# B&R Automation Studio project vibratorControlWithCurrentController (part 12)

#### producing.st
```iecst
ACTION producing:

	CASE em.state OF

		STATE_STOPPED:

			interface.status.ready 	:= FALSE;
			interface.status.active := TRUE; // need to tell wing when we are active. (otherwise wing start too fast and this task is stuck in STATE_ACTIVATING doing boot)

			em.cmd.sc 				:= TRUE;

		STATE_RESETTING:

			em.cmd.sc := TRUE;

		STATE_IDLE:
			interface.status.ready := TRUE;
			em.cmd.sc := TRUE;

		STATE_STARTING:

			interface.status.ready 									:= TRUE;
			interface.cmd.start										:= FALSE;
			interface.status.readyForStatusChange 					:= TRUE;
			this.cycleTime 											:= 0;
			em.cmd.sc 												:= TRUE;

		STATE_EXECUTE:

			CASE em.substate OF
				0: // H010 (Initialisation) + H020 (FM Start)
					em.cmd.sc := TRUE;
					interface.status.ready	:= TRUE;

					em.description := 'waiting for start command';
					IF interface.cmd.start THEN
						this.calculateCycletime := TRUE;
						IF interface.parameter.brickStatus = BRICK_STATUS_OK THEN
							this.MTDataStatistics_Real.Enable				:= TRUE;
							this.MTDataStatistics_Real.MovingWindowLength 	:= 10;
							this.MTDataStatistics_Real.In 					:= this.cycleTimeReal / 1000;
							this.MTDataStatistics_Real();
							this.cycleTimeReal := 0;
							IF this.MTDataStatistics_Real.Mean <> 0 THEN
								this.hmi.realMeanOutput := 60000 / this.MTDataStatistics_Real.Mean;
							END_IF
						END_IF

						// calculate cycletime here
						interface.cmd.start 						:= FALSE;
						interface.status.ready 						:= FALSE;
						this.time.elapsed							:= 0;
						this.time.maximum							:= interface.parameter.fallTime;
						gBottomFlapInterface.parameter.brickStatus 	:= interface.parameter.brickStatus;
						gBottomFlapInterface.cmd.brickStatusReady	:= TRUE;
						this.middleFlapTime 						:= 0;
						em.substate 								:= 40;
					ELSIF interface.cmd.manuelMode THEN
						em.substate := 1000;
					END_IF

				40: // H040 (FB Ready)
					em.description := 'waiting for bottom flap ready1 or ready2';

					this.time.elapsed := this.time.elapsed + em.status.cycleTime;

					IF gBottomFlapInterface.status.ready1 THEN
						interface.status.readyForStatusChange 		:= FALSE;
						gBottomFlapInterface.cmd.brickStatusReady	:= FALSE;
						gBottomFlapInterface.cmd.start1	:= TRUE;
						//em.cmd.sc := FALSE;
					END_IF

					// Wait FallTime before giving start2 (ok to give start1 before)
					IF gBottomFlapInterface.status.ready2 THEN
						em.cmd.sc := FALSE;
						this.flap.open := TRUE;
						this.cycleTimeTheoretical := 0;
						this.middleFlapTime := this.middleFlapTime + em.status.cycleTime;
						em.substate 			:= 70;
					END_IF

				70: // H070 (Open FM)
					em.description 				:= 'waiting for flap to be open';

					this.middleFlapTime := this.middleFlapTime + em.status.cycleTime;

					IF this.flap.error THEN
						this.alarm.openTooLong.active := TRUE;
						this.previousState := em.substate;
						em.substate := 700; // Error state in execute
					ELSIF this.flap.position = FLAP_OPEN THEN
						this.time.elapsed				:= 0;
						this.time.maximum				:= interface.parameter.openTime;
						gBottomFlapInterface.cmd.start2 := TRUE;
						interface.status.lastCycleTime 	:= UDINT_TO_REAL(this.middleFlapTime);
						interface.status.openCloseTime := this.cycleTimeTheoretical;
						em.substate 					:= 75;
					END_IF

				75: // H075
					em.description := 'waiting for opening time';

					this.middleFlapTime := this.middleFlapTime + em.status.cycleTime;
					this.time.elapsed	:= this.time.elapsed + em.status.cycleTime;

					IF this.time.elapsed >= this.time.maximum THEN
						this.flap.close := TRUE;
						em.substate := 80;
					END_IF

				80: // H080 (Close FM)
					em.description 				:= 'waiting for flap to be closed';

					this.middleFlapTime := this.middleFlapTime + em.status.cycleTime;

					IF this.flap.error THEN
						this.alarm.closeTooLong.active := TRUE;
						this.previousState := em.substate;
						em.substate := 700; // Error state in execute
					ELSIF this.flap.position = FLAP_CLOSED THEN
						interface.status.ready	:= TRUE;
						// Save open/close time in service menu (better than writing it cyclically).
						this.flapTest.openTime := this.flap.openTimeAfterChangeover;
						this.flapTest.closingTime := this.flap.closingTimeAfterChangeover;
						this.flapTest.openTimeOK := this.flapTest.openTime >= 210 AND this.flapTest.openTime <= 230;
						this.flapTest.closingTimeOK := this.flapTest.closingTime >= 210 AND this.flapTest.closingTime <= 230;
						this.cycleTime 			:= 0;
						this.hmi.portionCycleTime := UDINT_TO_REAL(this.middleFlapTime+gUpperFlapInterface.status.lastCycleTime)/1000;
						em.substate 			:= 0;
					END_IF

					(**** ERROR handling in EXECUTE ****)

				700:
					interface.cmd.runFlapContinuously	:= FALSE;
					interface.cmd.open					:= FALSE;
					interface.cmd.manuelMode			:= FALSE;

					IF NOT this.flap.error THEN
						this.flap.close := TRUE;
						em.substate := 710;
					ELSE
						this.flap.resetError := TRUE;
					END_IF

				710:
					em.description := 'Wait for flap to close - if not still continue. We cant be stuck in "SUSPENDING"';

					IF this.flap.error THEN
						this.time.elapsed := 0;
						em.substate := 720;
					ELSIF this.flap.position = FLAP_CLOSED THEN
						this.time.elapsed := 0;
						em.substate := 720;
					END_IF

				720:
					em.description := 'Wait for alarm acknowledge';

					this.time.elapsed := this.time.elapsed + em.status.cycleTime;

					IF this.time.elapsed >= 500000 THEN //500ms
						this.time.elapsed := 0;
						IF NOT MpAlarmXCheckReaction(mpAlarmXCore,'abortMain') THEN
							em.substate := 730; // "UNSUSPENDING"
						END_IF
					END_IF

				730:
					IF NOT this.flap.error THEN
						brsmemset(ADR(this.alarm), 0, SIZEOF(this.alarm));
						this.alarm.closeTooLong.name := 'middleFlapCloseTooLong';
						this.alarm.openTooLong.name := 'middleFlapOpenTooLong';
						this.flap.close := TRUE;
						em.substate := 740;
					ELSE
						this.flap.resetError := TRUE;
					END_IF

				740:
					em.description := 'Wait for flap to close -> if not go back and try again ';

					IF this.flap.error THEN
						em.substate := 730; // Try again (we MUST close flap before we return)
					ELSIF this.flap.position = FLAP_CLOSED THEN
						em.substate := 750;
					END_IF

				750:
					em.description := 'Recover to "previousState"';

					CASE this.previousState OF

						70: // Error opening
							em.cmd.sc := FALSE;
							this.flap.open := TRUE;
							this.cycleTimeTheoretical := 0;
							em.substate 			:= 70;

						80: // Error closing
							this.flap.close := TRUE;
							em.substate := 80;

						1000:
							em.substate := 0;

					END_CASE

					(**** Manuel mode ****)

				1000:
					testing;
					IF this.flap.error THEN
						// Stop testing and go in execute error state.
						this.previousState := em.substate;
						this.test.state := 0;

						em.substate := 700;
					END_IF

			END_CASE

			IF gMainInterface.status.state = STATE_EXECUTE THEN
				// calculate throughput cycletime
				this.cycleTime := this.cycleTime + UDINT_TO_REAL(em.status.cycleTime);
				this.cycleTimeReal := this.cycleTimeReal + UDINT_TO_REAL(em.status.cycleTime);
			ELSE
				this.MTDataStatistics_Real.Enable := FALSE;
				this.MTDataStatistics_Real();
				this.calculateCycletime := FALSE;
				this.cycleTime := 0;
				this.cycleTimeReal := 0;
				this.hmi.realMeanOutput := 0;
			END_IF

			this.cycleTimeTheoretical := this.cycleTimeTheoretical + em.status.cycleTime;

		STATE_COMPLETING:

			em.description := 'waiting for bottom flap ready2 to be ready';

			CASE em.substate OF

				0:
					// Determine if big or small brick from capcon teach integral
					IF gCapconInterface.status.teachIntegral > ELEMENT_SIZE_LIMIT AND gCapconInterface.status.teachingDone THEN
						this.ItemSize := Large;
					ELSE
						this.ItemSize := Small;
					END_IF

					em.substate := 10;

				10:
					IF gBottomFlapInterface.status.ready2 THEN
						gBeltInterface.cmd.stopDoingEmpty := FALSE;
						em.cmd.sc := TRUE;
					END_IF

			END_CASE

			em.setup.reactTo := BRDK_EM_REACT_TO_ALL;

		STATE_COMPLETE:

			CASE em.substate OF

				0:
					em.description 		:= 'empty or small items empty';

					IF this.ItemSize=Small THEN
						this.time.maximum := TIME_EMPTY_SMALL_ITEM;
						em.cmd.sc := FALSE;
						em.substate := 5;
					ELSE
						this.flap.open := TRUE;
						em.substate := 10;
						em.cmd.sc := TRUE;
					END_IF

				5:
					interface.status.ready := TRUE;
					em.description 		:= 'waiting for empty small items time or empty finished';
					this.time.elapsed	:= this.time.elapsed + em.status.cycleTime;

					IF this.time.elapsed >= this.time.maximum OR gMainInterface.status.state <> STATE_COMPLETING THEN
						interface.status.busy 	:= TRUE;
						this.time.elapsed 	:= 0;
						this.flap.open := TRUE;
						em.cmd.sc := FALSE;
						gBeltInterface.cmd.stopDoingEmpty := TRUE;
						em.substate 			:= 10;
					END_IF

					IF this.time.elapsed >= (this.time.maximum-400000) THEN
						// Signal belt and vibrator to stop 0.4s before opening flap.
						gBeltInterface.cmd.stopDoingEmpty := TRUE;
					END_IF

				10: // H820 (FM open)
					em.description 			:= 'waiting for flap to be open';

					IF this.flap.error THEN
						this.alarm.openTooLong.active := TRUE;
						this.previousState := em.substate;
						em.substate := 700; // Error state in execute
					ELSIF this.flap.position = FLAP_OPEN THEN
						this.time.elapsed				:= 0;
						this.time.maximum				:= 1000000; // 1s. be open for a longer time because a lot of bricks is falling and we dont want to pierce them.
						em.cmd.sc := TRUE;

						IF this.ItemSize=Small THEN
							em.substate 					:= 20;
						ELSE
							em.substate 					:= 40;
						END_IF

					END_IF

				20: //
					em.description 		:= 'waiting for opening time';
					this.time.elapsed	:= this.time.elapsed + em.status.cycleTime;

					IF this.time.elapsed >= this.time.maximum THEN
						this.flap.close := TRUE;
						em.cmd.sc := FALSE;
						interface.status.busy 			:= FALSE;
						em.substate 					:= 30;
					END_IF

				30: // H830 (FM close)
					em.description 		:= 'waiting for flap to be closed';

					IF this.flap.error THEN
						this.alarm.closeTooLong.active := TRUE;
						this.previousState := em.substate;
						em.substate := 700; // Error state in execute
					ELSIF this.flap.position = FLAP_CLOSED THEN
						interface.status.ready	:= TRUE;
						gBeltInterface.cmd.stopDoingEmpty := FALSE;
						this.flapTest.openTime := this.flap.openTimeAfterChangeover;
						this.flapTest.closingTime := this.flap.closingTimeAfterChangeover;
						this.flapTest.openTimeOK := this.flapTest.openTime >= 210 AND this.flapTest.openTime <= 230;
						this.flapTest.closingTimeOK := this.flapTest.closingTime >= 210 AND this.flapTest.closingTime <= 230;
						em.substate 			:= 0;
					END_IF

				40:
					em.description 		:= 'Emptying machine';
					interface.status.ready := TRUE;

						(**** ERROR handling in COMPLETE ****)

				700:
					interface.cmd.runFlapContinuously	:= FALSE;
					interface.cmd.open					:= FALSE;
					interface.cmd.manuelMode			:= FALSE;

					IF NOT this.flap.error THEN
						this.flap.close := TRUE;
						em.substate := 710;
					ELSE
						this.flap.resetError := TRUE;
					END_IF

				710:
					em.description := 'Wait for flap to close - if not still continue. We cant be stuck in "SUSPENDING"';

					IF this.flap.error THEN
						this.time.elapsed := 0;
						em.substate := 720;
					ELSIF this.flap.position = FLAP_CLOSED THEN
						this.time.elapsed := 0;
						em.substate := 720;
					END_IF

				720:
					em.description := 'Wait for alarm acknowledge';

					this.time.elapsed := this.time.elapsed + em.status.cycleTime;

					IF this.time.elapsed >= 500000 THEN //500ms
						this.time.elapsed := 0;
						IF NOT MpAlarmXCheckReaction(mpAlarmXCore,'abortMain') THEN
							em.substate := 730; // "UNSUSPENDING"
						END_IF
					END_IF

				730:
					IF NOT this.flap.error THEN
						brsmemset(ADR(this.alarm), 0, SIZEOF(this.alarm));
						this.alarm.closeTooLong.name := 'middleFlapCloseTooLong';
						this.alarm.openTooLong.name := 'middleFlapOpenTooLong';
						this.flap.close := TRUE;
						em.substate := 740;
					ELSE
						this.flap.resetError := TRUE;
					END_IF

				740:
					em.description := 'Wait for flap to close -> if not go back and try again ';

					IF this.flap.error THEN
						em.substate := 730; // Try again (we MUST close flap before we return)
					ELSIF this.flap.position = FLAP_CLOSED THEN
						em.substate := 750;
					END_IF

				750:
					em.description := 'Recover to "previousState"';

					CASE this.previousState OF

						10: // Error opening
							em.substate 			:= 0;

						30: // Error closing
							this.time.elapsed := 0;
							this.time.maximum := interface.parameter.openTime;
							em.substate := 20;

					END_CASE

		END_CASE

			gBottomFlapInterface.cmd.start1 := em.cmd.sc;

	STATE_ABORTED, STATE_SUSPENDED:
			em.description := 'waiting for wing to start';
			em.cmd.sc := TRUE;

	STATE_STOPPING, STATE_ABORTING, STATE_SUSPENDING:

			CASE em.substate OF

				0:
					em.description 				:= 'Clear status and close flap';
					interface.status.ready 					:= FALSE;
					interface.status.readyForStatusChange 	:= FALSE;
					interface.cmd.start 					:= FALSE;
					this.hw.do_open 		:= FALSE;
					interface.cmd.runFlapContinuously	:= FALSE;
					interface.cmd.open					:= FALSE;
					interface.cmd.manuelMode			:= FALSE;
					gBeltInterface.cmd.stopDoingEmpty := FALSE;

					IF NOT this.flap.error THEN
						this.flap.close := TRUE;
						em.substate := 10;
					ELSE
						this.flap.resetError := TRUE;
					END_IF

				10:
					em.description := 'Wait for flap to close';

					IF this.flap.error THEN
						em.substate := 20;
					ELSIF this.flap.position = FLAP_CLOSED THEN
						em.substate := 20;
					END_IF

				20:
					em.cmd.sc := TRUE;

			END_CASE

	STATE_CLEARING, STATE_UNSUSPENDING:
		em.description := 'waiting for flap error reset';

			CASE em.substate OF

				0:
					IF NOT this.flap.error THEN
						brsmemset(ADR(this.alarm), 0, SIZEOF(this.alarm));
						this.alarm.closeTooLong.name := 'middleFlapCloseTooLong';
						this.alarm.openTooLong.name := 'middleFlapOpenTooLong';
						this.flap.close := TRUE;
						em.substate := 10;
					ELSE
						this.flap.resetError := TRUE;
					END_IF

				10:
					em.description := 'Wait for flap to close';

					IF this.flap.error THEN
						em.substate := 0;
					ELSIF this.flap.position = FLAP_CLOSED THEN
						em.substate := 20;
					END_IF

				20:
					em.description 				:= 'Wait for close of own and neigbourflap';
					em.cmd.sc := TRUE;

			END_CASE

	ELSE
	em.cmd.sc := TRUE;

	END_CASE

END_ACTION
```

#### alarm.st
```iecst
ACTION alarm:

	// Open Time Too Long

	IF this.alarm.openTooLong.active AND NOT this.alarm.openTooLong.oldActive THEN
		this.alarm.openTooLong.instanceID := MpAlarmXSet(mpAlarmXCore, this.alarm.openTooLong.name);
	END_IF
	this.alarm.openTooLong.oldActive := this.alarm.openTooLong.active;

	// Close Time Too Long

	IF this.alarm.closeTooLong.active AND NOT this.alarm.closeTooLong.oldActive THEN
		this.alarm.closeTooLong.instanceID := MpAlarmXSet(mpAlarmXCore, this.alarm.closeTooLong.name);
	END_IF
	this.alarm.closeTooLong.oldActive := this.alarm.closeTooLong.active;

END_ACTION
```

#### middleFlap.st - Init, cyclic, exit code
```iecst
PROGRAM _INIT

	em.setup.name 			:= 'middleFlap';
	em.setup.parent.name 	:= 'wing';
	em.setup.reactTo 		:= BRDK_EM_REACT_TO_ALL;

	setupPointers;

	this.alarm.closeTooLong.name := 'middleFlapCloseTooLong';
	this.alarm.openTooLong.name := 'middleFlapOpenTooLong';

END_PROGRAM

PROGRAM _CYCLIC

	setupPointers;
	ioMappingInput;

	// setup flap function block
	this.flap.enable				:= TRUE;
	this.flap.cycleTime				:= em.status.cycleTime;
	this.flap.flapTime				:= interface.parameter.flapTime;
	this.flap.di_changeover 		:= this.hw.di_changeover;
	this.flap.simulation := gWingInterface.parameter.simulation;

	CASE em.mode OF
		MODE_PRODUCING,MODE_EMPTY: producing;
		MODE_MANUAL: testing;	// mode for testing flaps manually.
		ELSE em.cmd.sc := TRUE;
	END_CASE

	this.hw.do_open := this.flap.do_open;

	alarm;

	em();
	this.flap();

	// FAT test
	CASE testStateFAT OF

		0:
			IF interface.cmd.wingTestManual THEN
				// Only execute if flap is closed
				IF this.hw.do_open=FALSE THEN
					interface.status.testResultFAT := FALSE; // reset result
					testStateFAT := 10;
				END_IF

			END_IF

		10:
			//wait 1s so flaps are closed before we start test.
			this.TON_test.IN := TRUE;
			this.TON_test.PT := T#500ms;
			this.TON_test();

			IF this.TON_test.Q THEN
				this.TON_test.IN := FALSE;
				this.TON_test();

				// Open flap
				this.flap.open := TRUE;
				testStateFAT := 20;
			END_IF

		20:
			IF this.flap.error THEN
				// Test fail
				testStateFAT := 60;
			ELSIF this.flap.position = FLAP_OPEN THEN
				testStateFAT 			:= 30;
			END_IF

		30:
			//wait 1s before closing
			this.TON_test.IN := TRUE;
			this.TON_test.PT := T#500ms;
			this.TON_test();

			IF this.TON_test.Q THEN
				this.TON_test.IN := FALSE;
				this.TON_test();

				// Close flap
				this.flap.close := TRUE;
				testStateFAT := 40;
			END_IF

		40:
			IF this.flap.error THEN
				// Test fail
				testStateFAT := 60;
			ELSIF this.flap.position = FLAP_CLOSED THEN
				testStateFAT 			:= 50;
			END_IF

		50:
			//wait 1s before closing
			this.TON_test.IN := TRUE;
			this.TON_test.PT := T#500ms;
			this.TON_test();

			IF this.TON_test.Q THEN
				this.TON_test.IN := FALSE;
				this.TON_test();

				interface.status.testResultFAT := TRUE; // Good result
				testStateFAT := 60;
			END_IF

		60:
			// Reset error (if any) before finishing test
			this.flap.resetError := this.flap.error;

			IF NOT this.flap.error THEN
				interface.cmd.wingTestManual := FALSE; // signal test done

				// Start next test (we are done here)
				gBottomFlapInterface.cmd.wingTestManual := TRUE;
				testStateFAT := 0;
			END_IF

	END_CASE

END_PROGRAM

PROGRAM _EXIT

END_PROGRAM
```

#### ioMappingInput.st
```iecst
ACTION ioMappingInput:

	IF this.hwWu[0].di_wingUnitActive THEN
		this.flap.WUstepperConnected 	:= TRUE;
		this.flap.positionFromWUstepper	:= this.hwWu[0].flapPosition;
	ELSIF this.hwWu[1].di_wingUnitActive THEN
		this.flap.WUstepperConnected 	:= TRUE;
		this.flap.positionFromWUstepper	:= this.hwWu[1].flapPosition;
	ELSE
		this.flap.WUstepperConnected := FALSE;
	END_IF

END_ACTION
```

#### testing.st
```iecst
ACTION testing:

	this.flapTest.openTime := this.flap.openTimeAfterChangeover;
	this.flapTest.closingTime := this.flap.closingTimeAfterChangeover;
	this.flapTest.openTimeOK := this.flapTest.openTime >= 210 AND this.flapTest.openTime <= 230;
	this.flapTest.closingTimeOK := this.flapTest.closingTime >= 210 AND this.flapTest.closingTime <= 230;

	CASE this.test.state OF

		0:
			IF NOT interface.cmd.manuelMode THEN
				interface.cmd.runFlapContinuously := FALSE;
				em.substate := 0; // go back to 0 (no more manuel mode)
			ELSIF gWingInterface.status.startTestSequence THEN
				interface.cmd.runFlapContinuously := FALSE; // can't run while doing test sequence.
				this.test.state := 10;
			ELSIF interface.cmd.runFlapContinuously THEN
				this.test.state := 60;
			END_IF

			(**** Run sequence ****)

		10:
			IF NOT gWingInterface.status.startTestSequence THEN
				this.test.state := 0;
			ELSIF interface.cmd.open THEN
				this.flap.open := TRUE;
				this.test.state := 20;
			END_IF

		20:

			IF this.flap.error THEN
				this.alarm.openTooLong.active := TRUE;
			ELSIF this.flap.position = FLAP_OPEN THEN
				this.time.elapsed := 0;
				this.test.state := 30;
			END_IF

		30:
			this.time.elapsed := this.time.elapsed + em.status.cycleTime;
			IF this.time.elapsed >= this.flapTest.waitTime THEN
				this.flap.close := TRUE;		// close cmd
				this.test.state := 40;
			END_IF

		40:
			IF this.flap.error THEN
				this.alarm.closeTooLong.active := TRUE;
			ELSIF this.flap.position = FLAP_CLOSED THEN
				this.time.elapsed := 0;
				this.test.state := 50;
			END_IF

		50:
			em.description := 'Wait delay before opening next flap';

			this.time.elapsed := this.time.elapsed + em.status.cycleTime;
			IF this.time.elapsed >= this.flapTest.waitTime THEN
				interface.cmd.open := FALSE;	// Will signal to wing that flap is done with open/close.
				this.test.state := 10;
			END_IF

			(**** Run continously ****)

		60:
			IF NOT interface.cmd.runFlapContinuously THEN
				this.test.state := 0;
			ELSE
				this.flap.open := TRUE;
				this.test.state := 70;
			END_IF

		70:
			IF this.flap.error THEN
				this.alarm.openTooLong.active := TRUE;
			ELSIF this.flap.position = FLAP_OPEN THEN
				this.time.elapsed := 0;
				this.test.state := 80;
			END_IF

		80:
			this.time.elapsed := this.time.elapsed + em.status.cycleTime;
			IF this.time.elapsed >= this.flapTest.waitTime THEN
				this.flap.close := TRUE;		// close cmd
				this.test.state := 90;
			END_IF

		90:
			IF this.flap.error THEN
				this.alarm.closeTooLong.active := TRUE;
			ELSIF this.flap.position = FLAP_CLOSED THEN
				this.time.elapsed := 0;
				this.test.state := 100;
			END_IF

		100:
			this.time.elapsed := this.time.elapsed + em.status.cycleTime;
			IF this.time.elapsed >= this.flapTest.waitTime THEN
				this.test.state := 60;
			END_IF

	END_CASE

END_ACTION
```

#### setupPointers.st
```iecst
ACTION setupPointers:
	interface ACCESS ADR(gMiddleFlapInterface);
END_ACTION
```

#### local.typ - Local data types
```iecst
TYPE
	local_typ : 	STRUCT
		hw : local_hw_typ;
		hwAir : local_hw_typ;
		hwWu : ARRAY[0..1]OF wu20_typ; (*Communication with wing unit*)
		alarm : local_alarm_typ;
		time : local_time_typ;
		flap : legoCM20Flap;
		flapTest : flapTest_typ;
		MTDataStatistics_Real : MTDataStatistics;
		cycleTime : REAL;
		calculateCycletime : BOOL;
		hmi : local_hmi_typ;
		cycleTimeReal : REAL;
		cycleTimeTheoretical : UDINT;
		test : local_test_typ;
		previousState : UINT;
		middleFlapTime : UDINT;
		ItemSize : ITEM_SIZE_enum;
		TON_test : TON;
	END_STRUCT;
	ITEM_SIZE_enum :
		( (*Default large*)
		Large := 0,
		Small := 1
		);
	wu20_typ : 	STRUCT
		flapPosition : DINT; (*4 = open, 8 = closed*)
		di_wingUnitActive : BOOL;
	END_STRUCT;
	local_hmi_typ : 	STRUCT
		realMeanOutput : REAL;
		cycleTimeRaw : REAL;
		portionCycleTime : REAL;
	END_STRUCT;
	local_hw_typ : 	STRUCT
		di_changeover : BOOL;
		do_open : BOOL;
	END_STRUCT;
	local_alarm_typ : 	STRUCT
		openTooLong : gAlarm_struct_typ;
		closeTooLong : gAlarm_struct_typ;
	END_STRUCT;
	flapTest_typ : 	STRUCT
		flapSequenceTest : BOOL; (*Flaps will run in a sequence (usually over night)*)
		openTime : UDINT;
		closingTime : UDINT;
		waitTime : UDINT := 200000;
		alarmOpenTooLong : BOOL;
		alarmCloseTooLong : BOOL;
		openTimeOK : BOOL;
		closingTimeOK : BOOL;
	END_STRUCT;
	local_test_typ : 	STRUCT
		state : USINT;
	END_STRUCT;
END_TYPE
```

#### local.var - Local variables
```iecst
VAR CONSTANT
	ELEMENT_SIZE_LIMIT : REAL := 250000;
	TIME_EMPTY_SMALL_ITEM : UDINT := 20000000; (*20s*)
END_VAR
VAR
	interface : REFERENCE TO gMiddleFlapInterface_typ;
	this : {REDUND_UNREPLICABLE} local_typ;
	em : {REDUND_UNREPLICABLE} brdkEM;
	testStateFAT : USINT;
END_VAR
```

### middleFlapGlobal.var
```iecst
VAR
	gMiddleFlapInterface : gMiddleFlapInterface_typ;
END_VAR
```

### middleFlapGlobal.typ
```iecst
TYPE
	gMiddleFlapInterface_status_typ : 	STRUCT
		ready : BOOL;
		readyForStatusChange : BOOL;
		busy : BOOL;
		waitingForBottomOrCassette : BOOL;
		openCloseTime : UDINT;
		active : BOOL;
		lastCycleTime : REAL;
		testResultFAT : BOOL; (*TRUE=good, FALSE=bad*)
	END_STRUCT;
	gMiddleFlapInterface_para_typ : 	STRUCT
		brickStatus : gFlap_brick_status_typ;
		openTime : UDINT; (*Time the flap stays open*)
		flapTime : UDINT; (*Time that the flap is to open or close*)
		fallTime : UDINT; (*Time that a brick is to fall and be steady*)
		emptySmallItemsTime : UDINT; (*Time for flipping the flap when emptying small items*)
	END_STRUCT;
	gMiddleFlapInterface_cmd_typ : 	STRUCT
		start : BOOL;
		smallBrick : BOOL;
		updateStatistics : BOOL;
		runFlapContinuously : BOOL;
		open : BOOL; (*wing -> flap to open doing sequence test*)
		manuelMode : BOOL;
		wingTestManual : BOOL;
	END_STRUCT;
	gMiddleFlapInterface_typ : 	STRUCT
		cmd : gMiddleFlapInterface_cmd_typ;
		parameter : gMiddleFlapInterface_para_typ;
		status : gMiddleFlapInterface_status_typ;
	END_STRUCT;
END_TYPE
```

### Program Logical/modules/main/wing/bottomFlap/bottomFlap (IEC)

#### producing.st
```iecst
ACTION producing:

	CASE em.state OF

		STATE_STOPPED:

			interface.status.ready1 	:= FALSE;
			interface.status.ready2 	:= FALSE;
			interface.status.active := TRUE; // need to tell wing when we are active. (otherwise wing start too fast and this task is stuck in STATE_ACTIVATING doing boot)

			em.cmd.sc 					:= TRUE;

		STATE_RESETTING:

			em.cmd.sc := TRUE;

		STATE_IDLE:

			interface.status.ready1 := TRUE;
			em.cmd.sc 					:= TRUE;

		STATE_STARTING:

			interface.status.ready1 := TRUE;
			interface.cmd.start1	:= FALSE;
			interface.status.ready2 := FALSE;
			interface.cmd.start2	:= FALSE;
			em.cmd.sc 				:= TRUE;

		STATE_EXECUTE:

//			// Send to main -> ready to empty
//			IF gMainInterface.status.emptying THEN
//				// Only allow to empty if no brick in bottomFlap.
//				interface.status.emptyReady := em.substate < 110  OR em.substate >= 500 AND em.substate < 700;
//				em.cmd.sc := interface.status.emptyReady;
//			END_IF

			CASE em.substate OF

				0:	// I010 (Initialisation) + I020 (Bottom flap)
					em.description := 'waiting for start1 command';
					em.cmd.sc := TRUE;

					interface.status.ready1 := TRUE;

					interface.status.emptyReady := gMainInterface.status.emptying;

					IF interface.cmd.start1 AND NOT gMainInterface.status.emptying  THEN // added NOT emptying because otherwise wing could signal ".empty ready" and by the time main is going into completing em.substate is >=150 which till set em.cmd.sc=false. This will make bottom unable to follow main and freeze the machine

						em.cmd.sc 	:= FALSE;
						interface.cmd.start1	:= FALSE;
						interface.status.ready1 := FALSE;
						this.bottomFlapTime := 0;
						interface.status.emptyReady := FALSE;
						CASE interface.parameter.brickStatus OF

							BRICK_STATUS_OK:

								this.localShaftMode := interface.parameter.shaftMode;
								em.substate := 100;

							BRICK_STATUS_NOK:

								this.flap.open := TRUE;
								em.substate 			:= 400;				// Go to I400 (NOK)

						END_CASE

					END_IF

				100:
					em.description := 'waiting for neighbour to have a portion ready';

					IF gMainInterface.status.emptying THEN
						this.WingSync_0.Cancel := TRUE;
						this.WingSync_0.Request := FALSE;
					ELSIF this.localShaftMode = SHAFT_MODE_NORMAL AND NOT this.WingSync_0.Request THEN
						this.WingSync_0.Request := gCassetteInterface.status.syncAck = gCassetteInterface.cmd.start;
					ELSIF this.localShaftMode = SHAFT_MODE_EMPTY AND NOT this.WingSync_0.Request THEN
						this.WingSync_0.Request := gCassetteInterface.status.ready AND (gCassetteInterface.status.startAck = gCassetteInterface.cmd.start);
					END_IF

					IF this.WingSync_0.Approved THEN
						this.WingSync_0.Request := FALSE;
						this.WingSync_0.Cancel := FALSE;
						interface.status.ready2 := TRUE;
						this.bottomFlapTime := this.bottomFlapTime + em.status.cycleTime;
						interface.status.approvedPortion := TRUE;
				//		this.runningAlone := this.hw.di_neigbourIsDosing OR NOT (this.hw.di_neighbourActive);
						em.substate := 110;
					ELSIF this.WingSync_0.CancelApproved THEN
						this.WingSync_0.Request := FALSE;
						this.WingSync_0.Cancel := FALSE;
						em.substate := 0;
					END_IF

				110:
					em.description := 'waiting for start2 command';
					this.bottomFlapTime := this.bottomFlapTime + em.status.cycleTime;
					IF interface.cmd.start2 THEN
						interface.cmd.start2 := FALSE;
						interface.status.ready2 := FALSE;

						this.time.maximum := interface.parameter.fallTime;
						this.time.elapsed := 0;

						em.substate := 112;
					END_IF

				112:
					em.description := 'waiting for fall time';

					this.bottomFlapTime := this.bottomFlapTime + em.status.cycleTime;

					this.time.elapsed	:= this.time.elapsed + em.status.cycleTime;
					IF this.time.elapsed >= this.time.maximum THEN
						em.substate := 120;
					END_IF

				120:
					em.description := 'waiting for cassette to be ready';

					IF gCassetteInterface.status.ready AND (gCassetteInterface.status.startAck = gCassetteInterface.cmd.start) THEN
						this.bottomFlapTime := this.bottomFlapTime + em.status.cycleTime;
						this.flap.open := TRUE;
						this.neighbourFlap.open := TRUE;
						this.time.elapsed := 0;
						this.time.maximum := interface.parameter.cassetteStartDelay;
						this.cycleTimeTheoretical := 0;
						em.substate 		:= 310;
					ELSE
						this.timeWaitForCasstte := (this.timeWaitForCasstte + em.status.cycleTime)/1000;
					END_IF

				310: // I310 (Flap actions)
					em.description := 'waiting for own and neighbour flap to open and cassette delay to run out';

					this.bottomFlapTime := this.bottomFlapTime + em.status.cycleTime; // Neighbour flap is set open instantly when dual mahcines are connected
					IF this.flap.error OR this.neighbourFlap.error THEN
						this.alarm.openTooLong.active := this.flap.error;
						this.alarm.openNeighbourTooLong.active := this.neighbourFlap.error;
						this.previousState := em.substate;
						em.substate := 700; // Error in EXECUTE
					ELSIF this.flap.position = FLAP_OPEN AND this.neighbourFlap.position = FLAP_OPEN THEN
						em.substate := 315;
					END_IF

				315:
					em.description := 'Wait cassetteStartDelay';

					this.time.elapsed := this.time.elapsed + em.status.cycleTime;
					this.bottomFlapTime := this.bottomFlapTime + em.status.cycleTime;

					IF this.time.elapsed >= this.time.maximum THEN
						gCassetteInterface.cmd.start 	:= gCassetteInterface.cmd.start + 1;
						interface.status.approvedPortion := FALSE;
						this.OeeCalc_0.GoodPortion := this.OeeCalc_0.GoodPortion + 1;
						this.time.maximum				:= interface.parameter.openTime;
						em.substate 					:= 320;
					END_IF

				320:  // I320 (Cassette start)
					em.description := 'waiting for opening time';

					this.time.elapsed := this.time.elapsed + em.status.cycleTime;
					this.bottomFlapTime := this.bottomFlapTime + em.status.cycleTime;

					// if time elapsed close flap
					IF this.time.elapsed >= this.time.maximum THEN
						this.flap.close := TRUE;
						this.neighbourFlap.close := TRUE;
						em.substate := 330;
					END_IF

				330: // I330 (Flap actions)
					em.description := 'waiting for own and neighbour flaps to be closed';

					this.bottomFlapTime := this.bottomFlapTime + em.status.cycleTime; // Neighbour flap is set close instantly when dual mahcines are connected

					IF this.flap.error OR this.neighbourFlap.error THEN
						this.alarm.closeTooLong.active := this.flap.error;
						this.alarm.closeNeighbourTooLong.active := this.neighbourFlap.error;
						this.previousState := em.substate;
						em.substate := 700; // Error in EXECUTE
					ELSIF (this.flap.position = FLAP_CLOSED) AND (this.neighbourFlap.position = FLAP_CLOSED) THEN
						interface.status.ready1 := TRUE;
						interface.status.openCloseTime := this.cycleTimeTheoretical;
						// Save open/close time in service menu (better than writing it cyclically).
						this.flapTest.openTime := (this.flap.openTimeAfterChangeover);
						this.flapTest.closingTime := (this.flap.closingTimeAfterChangeover);
						this.flapTest.openTimeOK := this.flapTest.openTime >= 150 AND this.flapTest.openTime <= 170;
						this.flapTest.closingTimeOK := this.flapTest.closingTime >= 220 AND this.flapTest.closingTime <= 250;

						this.flapTest.neighbourClosingTime := (this.neighbourFlap.closingTimeAfterChangeover);
						this.flapTest.neighbourOpenTime := (this.neighbourFlap.openTimeAfterChangeover);
						this.flapTest.neighbourOpenTimeOK := this.flapTest.neighbourOpenTime >= 150 AND this.flapTest.neighbourOpenTime <= 170;
						this.flapTest.neighbourClosingTimeOK := this.flapTest.neighbourClosingTime >= 220 AND this.flapTest.neighbourClosingTime <= 250;

						this.hmi.portionCycleTime := UDINT_TO_REAL(this.bottomFlapTime) / 1000;

						em.substate := 0;
					END_IF

					(*** REJECT / NOK ***)

				400: // I400 (NOK)
					em.description := 'waiting for flap to be open and start 2 command';

					IF this.flap.error THEN
						this.alarm.openTooLong.active := TRUE;
						this.previousState := em.substate;
						em.substate := 700; // Error in EXECUTE
					ELSIF this.flap.position = FLAP_OPEN THEN
						interface.status.ready2 := TRUE;
						em.substate 			:= 410;
					END_IF

				410: // I400 (NOK)
					em.description := 'waiting for start2 command';

					IF interface.cmd.start2 THEN
						interface.cmd.start2 	:= FALSE;
						interface.status.ready2 := FALSE;
						this.OeeCalc_0.BadPortion := this.OeeCalc_0.BadPortion + 1;
						this.time.elapsed := 0;
						this.time.maximum := interface.parameter.fallTime;
						em.substate				:= 415;
					END_IF

				415: // Wait fall time - 150ms
					em.description := 'wait fall time';

					this.time.elapsed := this.time.elapsed + em.status.cycleTime;

					IF this.time.elapsed >= this.time.maximum THEN
						this.flap.close := TRUE;
						em.substate := 420;
					END_IF

				420: // I420
					em.description := 'waiting for flap to be closed';

					IF this.flap.error THEN
						this.alarm.closeTooLong.active := TRUE;
						this.previousState := em.substate;
						em.substate := 700; // Error in EXECUTE
					ELSIF this.flap.position = FLAP_CLOSED THEN
						interface.status.ready1	:= TRUE;

						// Save open/close time in service menu (better than writing it cyclically).
						this.flapTest.openTime := (this.flap.openTimeAfterChangeover);
						this.flapTest.closingTime := (this.flap.closingTimeAfterChangeover);
						this.flapTest.openTimeOK := this.flapTest.openTime >= 150 AND this.flapTest.openTime <= 170;
						this.flapTest.closingTimeOK := this.flapTest.closingTime >= 220 AND this.flapTest.closingTime <= 250;
						em.substate 			:= 0;
					END_IF

					(**** ERROR handling in EXECUTE ****)

				700:
					interface.cmd.runFlapContinuously	:= FALSE;
					interface.cmd.open					:= FALSE;
					interface.cmd.manuelMode			:= FALSE;

					IF NOT this.flap.error AND NOT this.neighbourFlap.error THEN
						this.flap.close := TRUE;
						this.neighbourFlap.close := TRUE;
						em.substate := 710;
					ELSE
						this.flap.resetError := this.flap.error;
						this.neighbourFlap.resetError := this.neighbourFlap.error;
					END_IF

				710:
					em.description := 'Wait for flap to close - if not still continue. We cant be stuck in "SUSPENDING"';

					IF this.flap.error OR this.neighbourFlap.error THEN
						this.time.elapsed := 0;
						em.substate := 720;
					ELSIF this.flap.position = FLAP_CLOSED AND this.neighbourFlap.position = FLAP_CLOSED THEN
						this.time.elapsed := 0;
						em.substate := 720;
					END_IF

				720:
					em.description := 'Wait for alarm acknowledge';

					this.time.elapsed := this.time.elapsed + em.status.cycleTime;

					IF this.time.elapsed >= 500000 THEN //500ms
						this.time.elapsed := 0;
						IF NOT MpAlarmXCheckReaction(mpAlarmXCore,'abortMain') THEN
							em.substate := 730; // "UNSUSPENDING"
						END_IF
					END_IF

				730:
					IF NOT this.flap.error AND NOT this.neighbourFlap.error THEN
						brsmemset(ADR(this.alarm), 0, SIZEOF(this.alarm));
						this.alarm.openTooLong.name := 'bottomFlapOpenTooLong';
						this.alarm.closeTooLong.name := 'bottomFlapCloseTooLong';
						this.alarm.openNeighbourTooLong.name := 'neighbourBottomFlapOpenTooLong';
						this.alarm.closeNeighbourTooLong.name := 'neighbourBottomFlapCloseTooLong';
						this.alarm.neighbourNotActive.name := 'neighbourNotActive';
						this.flap.close := TRUE;
						this.neighbourFlap.close := TRUE;
						em.substate := 740;
					ELSE
						this.flap.resetError := this.flap.error;
						this.neighbourFlap.resetError := this.neighbourFlap.error;
					END_IF

				740:
					em.description := 'Wait for flap to close -> if not go back and try again ';

					IF this.flap.error OR this.neighbourFlap.error THEN
						em.substate := 730; // Try again (we MUST close flap before we return)
					ELSIF this.flap.position = FLAP_CLOSED AND this.neighbourFlap.position = FLAP_CLOSED THEN
						em.substate := 750;
					END_IF

				750:
					em.description := 'Recover to "previousState"';

					CASE this.previousState OF

						0:
							em.substate := 0;

						310: // error opening flap
							this.flap.open := TRUE;
							this.neighbourFlap.open := TRUE;
							this.time.elapsed := 0;
							this.time.maximum := interface.parameter.cassetteStartDelay;
							this.cycleTimeTheoretical := 0;
							em.substate 		:= 310;

						330: // error closing flap
							this.flap.close := TRUE;
							this.neighbourFlap.close := TRUE;
							em.substate := 330;

						400: // error opening flap doing reject
							this.flap.open := TRUE;
							em.substate := 400;				// Go to I400 (NOK)

						420: // error closing flap doing reject
							this.flap.close := TRUE;
							em.substate := 420;

					END_CASE

			END_CASE

			(**** Manuel mode ****)

			// Had to move manuel mode to its own state diagram.
			CASE this.manuelState OF

				0:
					IF interface.cmd.manuelMode THEN
						this.test.state := 0;
						this.manuelState := 10;
					END_IF

				10:
					testing;
					IF this.flap.error THEN
						// Stop testing and go in execute error state.
						this.previousState := em.substate;
						this.test.state := 0;
						this.manuelState := 222;
						em.substate := 700;
					END_IF

				222:
					IF em.substate < 700 THEN
						// error has been acknowledged
						this.manuelState := 0;
					END_IF

			END_CASE

			this.cycleTimeTheoretical := this.cycleTimeTheoretical + em.status.cycleTime;

		STATE_STOPPING:
			CASE em.substate OF
				0:
					em.description 				:= 'Clear status and close flaps';

					this.flap.close := TRUE;
					this.neighbourFlap.close := TRUE;

					em.substate := 10;

				10:
					em.description 				:= 'waiting for own and neighbour flaps to be closed';

					IF this.flap.error OR this.neighbourFlap.error THEN
						interface.status.ready1 			:= FALSE;
						interface.cmd.start1				:= FALSE;
						interface.status.ready2 			:= FALSE;
						interface.cmd.start2				:= FALSE;
						interface.cmd.brickStatusReady		:= FALSE;
						this.WingSync_0.Request 			:= FALSE;
						em.substate := 100;
					ELSIF this.flap.position = FLAP_CLOSED AND this.neighbourFlap.position = FLAP_CLOSED THEN
						interface.status.ready1 			:= FALSE;
						interface.cmd.start1				:= FALSE;
						interface.status.ready2 			:= FALSE;
						interface.cmd.start2				:= FALSE;
						interface.cmd.brickStatusReady		:= FALSE;
						this.WingSync_0.Request 			:= FALSE;

						em.cmd.sc := TRUE;
					END_IF

					(* Error in STOPPING (just reset error - this will auto close) *)

				100:
					IF NOT this.flap.error AND NOT this.neighbourFlap.error THEN
						em.cmd.sc := TRUE;
					ELSE
						this.flap.resetError := this.flap.error;
						this.neighbourFlap.resetError := this.neighbourFlap.error;
					END_IF

			END_CASE

		STATE_ABORTED, STATE_SUSPENDED:
			em.description := 'waiting for wing to start';
			em.cmd.sc := TRUE;

		STATE_ABORTING, STATE_SUSPENDING:

			CASE em.substate OF

				0:
					em.description 				:= 'Clear status and close flap';
					interface.status.ready1 			:= FALSE;
					interface.cmd.start1				:= FALSE;
					interface.status.ready2 			:= FALSE;
					interface.cmd.start2				:= FALSE;
					this.hw.do_neighbourPortionReady 	:= FALSE;
					interface.cmd.brickStatusReady		:= FALSE;
					interface.cmd.runFlapContinuously	:= FALSE;
					interface.cmd.open					:= FALSE;
					interface.cmd.manuelMode			:= FALSE;

					IF NOT this.flap.error THEN
						this.flap.close := TRUE;
						em.substate := 10;
					ELSE
						this.flap.resetError := TRUE;
					END_IF

				10:
					em.description := 'Wait for flap to close';

					IF this.flap.error THEN
						em.substate := 20;
					ELSIF this.flap.position = FLAP_CLOSED THEN
						em.substate := 20;
					END_IF

				20:
					em.description := 'sc=true';
					em.cmd.sc := TRUE;

			END_CASE

		STATE_COMPLETING:

			this.WingSync_0.Request := FALSE;

			CASE em.substate OF
				0:
					em.description 				:= 'Open flap';
					this.timeWaitForCasstte := 0;
					this.flap.open := TRUE;

					em.substate := 10;
				10:
					em.description 				:= 'waiting for own flaps to be open';

					IF this.flap.error OR this.neighbourFlap.error THEN
						this.alarm.openTooLong.active := this.flap.error;
						this.previousState := em.substate;
						em.substate := 700;
					ELSIF this.flap.position = FLAP_OPEN THEN
						interface.status.ready2 := TRUE;
						em.cmd.sc := TRUE;
					END_IF

					(**** ERROR handling in COMPLETE ****)

				700:
					interface.cmd.runFlapContinuously	:= FALSE;
					interface.cmd.open					:= FALSE;
					interface.cmd.manuelMode			:= FALSE;

					IF NOT this.flap.error AND NOT this.neighbourFlap.error THEN
						this.flap.close := TRUE;
						this.neighbourFlap.close := TRUE;
						em.substate := 710;
					ELSE
						this.flap.resetError := this.flap.error;
						this.neighbourFlap.resetError := this.neighbourFlap.error;
					END_IF

				710:
					em.description := 'Wait for flap to close - if not still continue. We cant be stuck in "SUSPENDING"';

					IF this.flap.error OR this.neighbourFlap.error THEN
						this.time.elapsed := 0;
						em.substate := 720;
					ELSIF this.flap.position = FLAP_CLOSED AND this.neighbourFlap.position = FLAP_CLOSED THEN
						this.time.elapsed := 0;
						em.substate := 720;
					END_IF

				720:
					em.description := 'Wait for alarm acknowledge';

					this.time.elapsed := this.time.elapsed + em.status.cycleTime;

					IF this.time.elapsed >= 500000 THEN //500ms
						this.time.elapsed := 0;
						IF NOT MpAlarmXCheckReaction(mpAlarmXCore,'abortMain') THEN
							em.substate := 730; // "UNSUSPENDING"
						END_IF
					END_IF

				730:
					IF NOT this.flap.error AND NOT this.neighbourFlap.error THEN
						brsmemset(ADR(this.alarm), 0, SIZEOF(this.alarm));
						this.alarm.openTooLong.name := 'bottomFlapOpenTooLong';
						this.alarm.closeTooLong.name := 'bottomFlapCloseTooLong';
						this.alarm.openNeighbourTooLong.name := 'neighbourBottomFlapOpenTooLong';
						this.alarm.closeNeighbourTooLong.name := 'neighbourBottomFlapCloseTooLong';
						this.alarm.neighbourNotActive.name := 'neighbourNotActive';
						this.flap.close := TRUE;
						this.neighbourFlap.close := TRUE;
						em.substate := 740;
					ELSE
						this.flap.resetError := this.flap.error;
						this.neighbourFlap.resetError := this.neighbourFlap.error;
					END_IF

				740:
					em.description := 'Wait for flap to close -> if not go back and try again ';

					IF this.flap.error OR this.neighbourFlap.error THEN
						em.substate := 730; // Try again (we MUST close flap before we return)
					ELSIF this.flap.position = FLAP_CLOSED AND this.neighbourFlap.position = FLAP_CLOSED THEN
						em.substate := 750;
					END_IF

				750:
					em.description := 'Recover to "previousState"';

					CASE this.previousState OF

						10: // Error opening
							this.flap.open := TRUE;
							em.substate := 0;

					END_CASE

			END_CASE;

		STATE_COMPLETE:
			em.description 				:= 'Emptying machine';
			em.setup.reactTo := BRDK_EM_REACT_TO_ALL;
			em.cmd.start := TRUE;

			IF interface.cmd.start1 THEN
				this.time.elapsed :=  this.time.elapsed + em.status.cycleTime;
			ELSE
				this.time.maximum := 1000000; // 1 sec
				this.time.elapsed := 0;
			END_IF

			em.cmd.sc :=  this.time.elapsed > this.time.maximum AND this.flap.position = FLAP_OPEN; // Flap must be open since we go to STATE_STOPPING and closes both flaps.

		STATE_CLEARING, STATE_UNSUSPENDING:

			CASE em.substate OF
				0:
					em.description 				:= 'Clear own status';
					interface.status.ready1 			:= FALSE;
					interface.cmd.start1				:= FALSE;
					interface.status.ready2 			:= FALSE;
					interface.cmd.start2				:= FALSE;
					this.hw.do_neighbourPortionReady 	:= FALSE;
					em.substate := 5;

				5:
					em.description 				:= 'Clear own flap error';
					IF NOT this.flap.error THEN
						brsmemset(ADR(this.alarm), 0, SIZEOF(this.alarm));
						// Alarm texts
						this.alarm.openTooLong.name := 'bottomFlapOpenTooLong';
						this.alarm.closeTooLong.name := 'bottomFlapCloseTooLong';
						this.alarm.openNeighbourTooLong.name := 'neighbourBottomFlapOpenTooLong';
						this.alarm.closeNeighbourTooLong.name := 'neighbourBottomFlapCloseTooLong';
						this.alarm.neighbourNotActive.name := 'neighbourNotActive';
						this.flap.close := TRUE;
						em.substate := 10;
					ELSE
						this.flap.resetError := TRUE;
					END_IF

				10:
					em.description := 'Wait for flap to close';

					IF this.flap.error THEN
						em.substate := 5;
					ELSIF this.flap.position = FLAP_CLOSED THEN
						em.substate := 20;
					END_IF

				20:
					em.description 				:= 'Wait for close of own and neigbourflap';
					em.cmd.sc := TRUE;

			END_CASE

		ELSE
			em.cmd.sc := TRUE;

	END_CASE

END_ACTION
```

#### alarm.st
```iecst
ACTION alarm:

	// Open Time Too Long

	IF this.alarm.openTooLong.active AND NOT this.alarm.openTooLong.oldActive THEN
		this.alarm.openTooLong.instanceID := MpAlarmXSet(mpAlarmXCore, this.alarm.openTooLong.name);
	END_IF
	this.alarm.openTooLong.oldActive := this.alarm.openTooLong.active;

	// Close Time Too Long

	IF this.alarm.closeTooLong.active AND NOT this.alarm.closeTooLong.oldActive THEN
		this.alarm.closeTooLong.instanceID := MpAlarmXSet(mpAlarmXCore, this.alarm.closeTooLong.name);
	END_IF
	this.alarm.closeTooLong.oldActive := this.alarm.closeTooLong.active;

	// Open Neighbour Time Too Long

	IF this.alarm.openNeighbourTooLong.active AND NOT this.alarm.openNeighbourTooLong.oldActive THEN
		this.alarm.openNeighbourTooLong.instanceID := MpAlarmXSet(mpAlarmXCore, this.alarm.openNeighbourTooLong.name);
	END_IF
	this.alarm.openNeighbourTooLong.oldActive := this.alarm.openNeighbourTooLong.active;

	// Close Neighbour Time Too Long

	IF this.alarm.closeNeighbourTooLong.active AND NOT this.alarm.closeNeighbourTooLong.oldActive THEN
		this.alarm.closeNeighbourTooLong.instanceID := MpAlarmXSet(mpAlarmXCore, this.alarm.closeNeighbourTooLong.name);
	END_IF
	this.alarm.closeNeighbourTooLong.oldActive := this.alarm.closeNeighbourTooLong.active;

	// Neighbour machine not active

	this.alarm.neighbourNotActive.active := NOT this.hw.di_neighbourActive AND this.old_neighbourActive AND gMainInterface.status.machineStart;
	this.old_neighbourActive := this.hw.di_neighbourActive;

	IF this.alarm.neighbourNotActive.active AND NOT this.alarm.neighbourNotActive.oldActive THEN
		this.alarm.neighbourNotActive.instanceID := MpAlarmXSet(mpAlarmXCore, this.alarm.neighbourNotActive.name);
		interface.status.neighbourDisappeared := TRUE;
	END_IF
	this.alarm.neighbourNotActive.oldActive := this.alarm.neighbourNotActive.active;

END_ACTION
```

#### bottomFlap.st - Init, cyclic, exit code
```iecst
PROGRAM _INIT

	em.setup.name 			:= 'bottomFlap';
	em.setup.parent.name 	:= 'wing';
	em.setup.reactTo 		:= BRDK_EM_REACT_TO_ALL;

	setupPointers;

	// Alarm texts
	this.alarm.openTooLong.name := 'bottomFlapOpenTooLong';
	this.alarm.closeTooLong.name := 'bottomFlapCloseTooLong';
	this.alarm.openNeighbourTooLong.name := 'neighbourBottomFlapOpenTooLong';
	this.alarm.closeNeighbourTooLong.name := 'neighbourBottomFlapCloseTooLong';
	this.alarm.neighbourNotActive.name := 'neighbourNotActive';

	cm20Connected := TRUE;

END_PROGRAM

PROGRAM _CYCLIC

	setupPointers;
	ioMappingInput;

	// this.runningAlone := this.hw.di_neigbourIsDosing OR NOT (this.hw.di_neighbourActive);

	// setup flap function block
	this.flap.enable 						 := TRUE;
	this.flap.cycleTime						 := em.status.cycleTime;
	this.flap.flapTime						 := interface.parameter.flapTime;
	this.flap.di_changeover 				 := this.hw.di_changeover;
	this.flap.simulation					 := gWingInterface.parameter.simulation;
	this.neighbourFlap.enable				 := NOT this.WingSync_0.RunningWithNeighbour;
	this.neighbourFlap.cycleTime			 := em.status.cycleTime;
	this.neighbourFlap.flapTime				 := interface.parameter.flapTime;
	this.neighbourFlap.di_changeover 		 := this.hw.di_neighbourChangeover;
	this.neighbourFlap.simulation			 := gWingInterface.parameter.simulation;

	this.flap();
	this.neighbourFlap();

	CASE em.mode OF
		MODE_PRODUCING: producing;
		MODE_MANUAL: testing;	// mode for testing flaps manually.
		ELSE em.cmd.sc := TRUE;
	END_CASE

	this.hw.do_open				:= this.flap.do_open;
	this.hw.do_neighbourOpen	:= this.neighbourFlap.do_open;
	this.hmi.neighbourActive	:= this.hw.di_neighbourActive;

	alarm;

	em();

	this.WingSync_0.NeighbourActive 			:= this.hw.di_neighbourActive;
	this.WingSync_0.NeighbourIsDosing 			:= this.hw.di_neigbourIsDosing;
	this.WingSync_0.di_neighbourPortionReady 	:= this.hw.di_neighbourPortionReady;
	this.WingSync_0();
	this.hw.do_neighbourPortionReady 			:= this.WingSync_0.do_neighbourPortionReady;

	this.OeeCalc_0.Enable := TRUE;
	this.OeeCalc_0.Executing := gMainInterface.status.state = STATE_EXECUTE;
	this.OeeCalc_0.IdealCycleTime := 1200;
	this.OeeCalc_0.Reset := gMainInterface.status.state = STATE_COMPLETING;
	this.OeeCalc_0();

	interface.status.waitingForNeighbour 		:= this.WingSync_0.WaitingForNeighbour;
	interface.status.neighbourWaiting			:= this.hw.di_neighbourPortionReady;

	// FAT test
	CASE testStateFAT OF

		0:
			IF interface.cmd.wingTestManual THEN
				// Only execute if flap is closed
				IF this.hw.do_open=FALSE AND this.hw.do_neighbourOpen=FALSE THEN
					interface.status.testResultFAT := FALSE; // reset result
					testStateFAT := 10;
				END_IF

			END_IF

		10:
			//wait 1s so flaps are closed before we start test.
			this.TON_test.IN := TRUE;
			this.TON_test.PT := T#500ms;
			this.TON_test();

			IF this.TON_test.Q THEN
				this.TON_test.IN := FALSE;
				this.TON_test();

				// Open flap
				this.flap.open := TRUE;
				testStateFAT := 20;
			END_IF

		20:
			IF this.flap.error THEN
				// Test fail
				testStateFAT := 120;
			ELSIF this.flap.position = FLAP_OPEN THEN
				testStateFAT 			:= 30;
			END_IF

		30:
			//wait 1s before closing
			this.TON_test.IN := TRUE;
			this.TON_test.PT := T#500ms;
			this.TON_test();

			IF this.TON_test.Q THEN
				this.TON_test.IN := FALSE;
				this.TON_test();

				// Close flap
				this.flap.close := TRUE;
				testStateFAT := 40;
			END_IF

		40:
			IF this.flap.error THEN
				// Test fail
				testStateFAT := 120;
			ELSIF this.flap.position = FLAP_CLOSED THEN
				testStateFAT 			:= 50;
			END_IF

		50:
			//wait 1s
			this.TON_test.IN := TRUE;
			this.TON_test.PT := T#500ms;
			this.TON_test();

			IF this.TON_test.Q THEN
				this.TON_test.IN := FALSE;
				this.TON_test();

				// start test of neighbourFlap
				this.neighbourFlap.open := TRUE;
				testStateFAT := 60;
			END_IF

		60:
			IF this.neighbourFlap.error THEN
				// test Fail
				testStateFAT := 120;
			ELSIF this.neighbourFlap.position = FLAP_OPEN THEN
				testStateFAT := 70;
			END_IF

		70:
			//wait 1s
			this.TON_test.IN := TRUE;
			this.TON_test.PT := T#500ms;
			this.TON_test();

			IF this.TON_test.Q THEN
				this.TON_test.IN := FALSE;
				this.TON_test();

				// start test of neighbourFlap
				this.neighbourFlap.close := TRUE;
				testStateFAT := 80;
			END_IF

		80:
			IF this.neighbourFlap.error THEN
				// test Fail
				testStateFAT := 120;
			ELSIF this.flap.position = FLAP_CLOSED THEN
				testStateFAT := 90;
			END_IF

		90:
			//wait 1s
			this.TON_test.IN := TRUE;
			this.TON_test.PT := T#500ms;
			this.TON_test();

			IF this.TON_test.Q THEN
				this.TON_test.IN := FALSE;
				this.TON_test();

				interface.status.testResultFAT := TRUE; // Good result
				testStateFAT := 120;
			END_IF

		120:
			// Reset error (if any) before finishing test
			this.flap.resetError := this.flap.error;
			this.neighbourFlap.resetError := this.neighbourFlap.error;

			IF NOT this.flap.error AND NOT this.neighbourFlap.error THEN
				interface.cmd.wingTestManual := FALSE; // signal test done

				// Start next test (we are done here)
				gCassetteInterface.cmd.wingTestManual := TRUE;
				testStateFAT := 0;
			END_IF

	END_CASE

END_PROGRAM

PROGRAM _EXIT

END_PROGRAM
```

#### ioMappingInput.st
```iecst
ACTION ioMappingInput:

	IF this.hwWu[0].di_wingUnitActive THEN
		this.hw.di_neigbourIsDosing				 := this.hwWu[0].neigbourIsDosing;
		this.hw.di_neighbourActive				 := this.hwWu[0].neighbourActive;
		this.hw.di_neighbourPortionReady		 := this.hwWu[0].neighbourPortionReady;
		this.flap.WUstepperConnected			 := TRUE;
		this.flap.positionFromWUstepper 		 := this.hwWu[0].flapPosition;
		this.neighbourFlap.WUstepperConnected	 := TRUE;
		this.neighbourFlap.positionFromWUstepper := this.hwWu[0].neighbourFlapPosition;
	ELSIF this.hwWu[1].di_wingUnitActive THEN
		this.hw.di_neigbourIsDosing				 := this.hwWu[1].neigbourIsDosing;
		this.hw.di_neighbourActive				 := this.hwWu[1].neighbourActive;
		this.hw.di_neighbourPortionReady		 := this.hwWu[1].neighbourPortionReady;
		this.flap.WUstepperConnected			 := TRUE;
		this.flap.positionFromWUstepper 		 := this.hwWu[1].flapPosition;
		this.neighbourFlap.WUstepperConnected	 := TRUE;
		this.neighbourFlap.positionFromWUstepper := this.hwWu[1].neighbourFlapPosition;
	ELSE
		this.hw.di_neigbourIsDosing				 := this.hwAir.di_neigbourIsDosing;
		this.hw.di_neighbourActive				 := this.hwAir.di_neighbourActive;
		this.hw.di_neighbourPortionReady		 := this.hwAir.di_neighbourPortionReady;
		this.flap.WUstepperConnected			 := FALSE;
	END_IF

END_ACTION
```

#### testing.st
```iecst
ACTION testing:

	this.flapTest.openTime := this.flap.openTimeAfterChangeover;
	this.flapTest.closingTime := this.flap.closingTimeAfterChangeover;
	this.flapTest.openTimeOK := this.flapTest.openTime >= 150 AND this.flapTest.openTime <= 170;
	this.flapTest.closingTimeOK := this.flapTest.closingTime >= 220 AND this.flapTest.closingTime <= 250;

	CASE this.test.state OF

		0:
			IF NOT interface.cmd.manuelMode THEN
				interface.cmd.runFlapContinuously := FALSE;
				this.manuelState := 0; // go back to 0 (no more manuel mode)
			ELSIF gWingInterface.status.startTestSequence THEN
				interface.cmd.runFlapContinuously := FALSE; // can't run while doing test sequence.
				this.test.state := 10;
			ELSIF interface.cmd.runFlapContinuously THEN
				this.test.state := 60;
			END_IF

		(**** Run sequence ****)

		10:
			IF NOT gWingInterface.status.startTestSequence THEN
				this.test.state := 0;
			ELSIF interface.cmd.open THEN
				this.flap.open := TRUE;
				this.test.state := 20;
			END_IF

		20:

			IF this.flap.error THEN
				this.alarm.openTooLong.active := TRUE;
			ELSIF this.flap.position = FLAP_OPEN THEN
				this.time.elapsed := 0;
				this.test.state := 30;
			END_IF

		30:
			this.time.elapsed := this.time.elapsed + em.status.cycleTime;
			IF this.time.elapsed >= this.flapTest.waitTime THEN
				this.flap.close := TRUE;		// close cmd
				this.test.state := 40;
			END_IF

		40:
			IF this.flap.error THEN
				this.alarm.closeTooLong.active := TRUE;
			ELSIF this.flap.position = FLAP_CLOSED THEN
				this.time.elapsed := 0;
				this.test.state := 50;
			END_IF

		50:
			em.description := 'Wait delay before opening next flap';

			this.time.elapsed := this.time.elapsed + em.status.cycleTime;
			IF this.time.elapsed >= this.flapTest.waitTime THEN
				interface.cmd.open := FALSE;	// Will signal to wing that flap is done with open/close.
				this.test.state := 10;
			END_IF

		(**** Run continously ****)

		60:
			IF NOT interface.cmd.runFlapContinuously THEN
				this.test.state := 0;
			ELSE
				this.flap.open := TRUE;
				this.test.state := 70;
			END_IF

		70:
			IF this.flap.error THEN
				this.alarm.openTooLong.active := TRUE;
			ELSIF this.flap.position = FLAP_OPEN THEN
				this.time.elapsed := 0;
				this.test.state := 80;
			END_IF

		80:
			this.time.elapsed := this.time.elapsed + em.status.cycleTime;
			IF this.time.elapsed >= this.flapTest.waitTime THEN
				this.flap.close := TRUE;		// close cmd
				this.test.state := 90;
			END_IF

		90:
			IF this.flap.error THEN
				this.alarm.closeTooLong.active := TRUE;
			ELSIF this.flap.position = FLAP_CLOSED THEN
				this.time.elapsed := 0;
				this.test.state := 100;
			END_IF

		100:
			this.time.elapsed := this.time.elapsed + em.status.cycleTime;
			IF this.time.elapsed >= this.flapTest.waitTime THEN
				this.test.state := 60;
			END_IF

	END_CASE

END_ACTION
```

#### setupPointers.st
```iecst
ACTION setupPointers:
	interface ACCESS ADR(gBottomFlapInterface);
END_ACTION
```

#### local.typ - Local data types
```iecst
TYPE
	local_typ : 	STRUCT
		alarm : local_alarm_typ;
		hw : local_hw_typ;
		hwAir : local_hw_typ;
		hwWu : ARRAY[0..1]OF wu20_typ;
		time : local_time_typ;
		neighbourFlap : legoCM20Flap;
		flap : legoCM20Flap;
		hmi : local_hmi_typ;
		flapTest : flapTest_typ;
		localShaftMode : gBottomShaftMode_typ;
		timeWaitForCasstte : UDINT; (*Only for statistics to see how long we wait for cassettes*)
		WingSync_0 : WingSync;
		old_neighbourActive : BOOL;
		cycleTimeTheoretical : UDINT;
		runningAlone : BOOL;
		test : local_test_typ;
		previousState : UINT;
		bottomFlapTime : UDINT;
		manuelState : USINT;
		OeeCalc_0 : OeeCalc;
		TON_test : TON;
	END_STRUCT;
	local_test_typ : 	STRUCT
		state : USINT;
	END_STRUCT;
	wu20_typ : 	STRUCT
		flapPosition : DINT; (*4 = open, 8 = closed*)
		neighbourFlapPosition : DINT; (*4 = open, 8 = closed*)
		neighbourActive : BOOL;
		neigbourIsDosing : BOOL;
		neighbourPortionReady : BOOL;
		di_wingUnitActive : BOOL;
	END_STRUCT;
	local_hmi_typ : 	STRUCT
		neighbourActive : BOOL;
		forceEmpty : BOOL; (*If operator force an empty even though we have a brick in bottom flap.*)
		portionCycleTime : REAL;
	END_STRUCT;
	local_hw_typ : 	STRUCT
		di_neighbourChangeover : BOOL;
		do_neighbourOpen : BOOL;
		di_changeover : BOOL;
		do_open : BOOL;
		di_neighbourPortionReady : BOOL; (*Signal name: DI_WU_NFMRDY
PJ95: WU_S
Connector: DI.16
Description: Signal from neighbour CM. �1� indicates elements are ready on neighbour middle flap. Utilized for synchronization shaft with neighbour CM. Only relevant if DI_WU_NCON is active.*)
		do_neighbourPortionReady : BOOL; (*Signal name: DO_WU_NFMRDY
PJ95: WU_S
Connector: DO.16
Description: Signal to neighbour CM. �1� means elements are ready on middle flap. Utilized for synchronization shaft with neighbour CM.*)
		di_neighbourActive : BOOL; (*Signal name: DI_WU_NCON
PJ95: WU_S
Connector: DI.18
Description: Signal from neighbour CM. �1� indicates a neighbour CM is connected and active.*)
		di_neigbourIsDosing : BOOL;
	END_STRUCT;
	local_alarm_typ : 	STRUCT
		openTooLong : gAlarm_struct_typ;
		closeTooLong : gAlarm_struct_typ;
		openNeighbourTooLong : gAlarm_struct_typ;
		closeNeighbourTooLong : gAlarm_struct_typ;
		neighbourNotActive : gAlarm_struct_typ;
	END_STRUCT;
	flapTest_typ : 	STRUCT
		flapSequenceTest : BOOL; (*Flaps will run in a sequence (usually over night)*)
		openTime : UDINT;
		closingTime : UDINT;
		neighbourOpenTime : UDINT;
		neighbourClosingTime : UDINT;
		waitTime : UDINT := 200000;
		alarmOpenTooLong : BOOL;
		alarmCloseTooLong : BOOL;
		openTimeOK : BOOL;
		closingTimeOK : BOOL;
		neighbourOpenTimeOK : BOOL;
		neighbourClosingTimeOK : BOOL;
	END_STRUCT;
END_TYPE
```

#### local.var - Local variables
```iecst
VAR
	cm20Connected : {REDUND_UNREPLICABLE} BOOL := TRUE;
	interface : REFERENCE TO gBottomFlapInterface_typ;
	this : {REDUND_UNREPLICABLE} local_typ;
	em : {REDUND_UNREPLICABLE} brdkEM;
END_VAR
VAR CONSTANT
	TRANSMISSION_DELAY : UDINT := 10000;
END_VAR
VAR
	testStateFAT : USINT;
END_VAR
```

#### LocalFunctions.fun
```iecst
FUNCTION_BLOCK OeeCalc
	VAR_INPUT
		Enable : BOOL;
	END_VAR
	VAR_INPUT RETAIN
		BadPortion : UDINT;
		GoodPortion : UDINT;
	END_VAR
	VAR_INPUT
		Executing : BOOL;
		IdealCycleTime : REAL;
		Reset : BOOL;
	END_VAR
	VAR_OUTPUT
		Active : BOOL;
		Availability : REAL;
		Performance : REAL;
		Quality : REAL;
		OEE : REAL;
	END_VAR
	VAR
		state : INT;
		RTInfo_0 : RTInfo;
	END_VAR
	VAR RETAIN
		executeTime : UDINT;
		totalTime : UDINT;
	END_VAR
END_FUNCTION_BLOCK

{REDUND_ERROR} FUNCTION_BLOCK WingSync (*Function block that handles synchronization between two CMs*) (*$GROUP=User,$CAT=User,$GROUPICON=User.png,$CATICON=User.png*)
	VAR_INPUT
		Request : BOOL; (*Request synchronization with neighbour machine*)
		di_neighbourPortionReady : BOOL;
		NeighbourActive : BOOL;
		NeighbourIsDosing : BOOL;
		Cancel : BOOL;
	END_VAR
	VAR_OUTPUT
		do_neighbourPortionReady : BOOL;
		Approved : BOOL; (*Syncronization with neighbour completed*)
		CancelApproved : BOOL;
		WaitingForNeighbour : BOOL;
		RunningWithNeighbour : BOOL;
	END_VAR
	VAR
		state : UINT;
		TON_transmissionDelay : TON;
		TON_timeout : TON;
	END_VAR
END_FUNCTION_BLOCK
```

#### LocalFunctions.st
```iecst
(* Function block that handles synchronization between two CMs *)
FUNCTION_BLOCK WingSync

	CASE state OF
		0:
			IF Request THEN
				IF NeighbourIsDosing THEN
					Approved := TRUE;
					RunningWithNeighbour := FALSE;
					state := 30;
				ELSE
					do_neighbourPortionReady := TRUE;
					state := 10;
				END_IF
			ELSIF Cancel THEN
				state := 220;
			END_IF

		10:
			IF di_neighbourPortionReady THEN
				state := 15;
			ELSIF NeighbourIsDosing THEN
				TON_timeout.IN := FALSE;
				TON_timeout();
				state := 300;
			ELSIF Cancel THEN
				TON_timeout.IN := FALSE;
				TON_timeout();
				state := 200;
			END_IF

		15:
			TON_transmissionDelay.IN := TRUE;
			TON_transmissionDelay.PT:= T#10ms;
			TON_transmissionDelay();

			IF TON_transmissionDelay.Q THEN
				TON_transmissionDelay.IN := FALSE;
				TON_transmissionDelay();
				do_neighbourPortionReady := FALSE;
				state := 20;
			END_IF

		20:
			IF NOT di_neighbourPortionReady THEN
				Approved := TRUE;
				RunningWithNeighbour := TRUE;
				state := 30;
			END_IF

		30:
			IF NOT Request THEN
				Approved := FALSE;
				state := 0;
			END_IF

		100:
			Approved := Request;
			CancelApproved := Cancel;
			RunningWithNeighbour := FALSE;

			IF NeighbourActive THEN
				Approved := FALSE;
				CancelApproved := FALSE;
				state := 0;
			END_IF

		200:
			do_neighbourPortionReady := FALSE;

			TON_timeout.IN := TRUE;
			TON_timeout.PT := T#100ms;
			TON_timeout();

			IF di_neighbourPortionReady THEN
				TON_timeout.IN := FALSE;
				TON_timeout();
				state := 210;
			ELSIF TON_timeout.Q THEN
				TON_timeout.IN := FALSE;
				TON_timeout();
				state := 220;
			END_IF

		210:
			TON_timeout.IN := TRUE;
			TON_timeout.PT := T#100ms;
			TON_timeout();

			IF NOT di_neighbourPortionReady THEN
				TON_timeout.IN := FALSE;
				TON_timeout();
				Approved := TRUE;
				RunningWithNeighbour := TRUE;
				state := 30;
			ELSIF TON_timeout.Q THEN
				TON_timeout.IN := FALSE;
				TON_timeout();
				state := 220;
			END_IF

		220:
			CancelApproved := TRUE;
			RunningWithNeighbour := FALSE;

			IF NOT Cancel THEN
				CancelApproved := FALSE;
				state := 0;
			END_IF

		300:
			do_neighbourPortionReady := FALSE;

			TON_timeout.IN := TRUE;
			TON_timeout.PT := T#100ms;
			TON_timeout();

			IF di_neighbourPortionReady THEN
				TON_timeout.IN := FALSE;
				TON_timeout();
				state := 310;
			ELSIF TON_timeout.Q THEN
				TON_timeout.IN := FALSE;
				TON_timeout();
				Approved := TRUE;
				RunningWithNeighbour := FALSE;
				state := 30;
			END_IF

		310:
			TON_timeout.IN := TRUE;
			TON_timeout.PT := T#100ms;
			TON_timeout();

			IF NOT di_neighbourPortionReady THEN
				TON_timeout.IN := FALSE;
				TON_timeout();
				Approved := TRUE;
				RunningWithNeighbour := TRUE;
				state := 30;
			ELSIF TON_timeout.Q THEN
				TON_timeout.IN := FALSE;
				TON_timeout();
				Approved := TRUE;
				RunningWithNeighbour := FALSE;
				state := 30;
			END_IF

	END_CASE

	WaitingForNeighbour := do_neighbourPortionReady AND NOT di_neighbourPortionReady;

	IF NOT NeighbourActive THEN
		do_neighbourPortionReady := FALSE;
		state := 100;
	END_IF

END_FUNCTION_BLOCK

FUNCTION_BLOCK OeeCalc

	IF NOT Enable AND Active THEN
		state := 0;
		Active := FALSE;
	END_IF

	CASE state OF
		0:
			IF Enable THEN
				Active := TRUE;
				state := 10;
			END_IF

		10:
			RTInfo_0.enable := TRUE;
			RTInfo_0();

			IF RTInfo_0.status = ERR_OK THEN
				state := 20;
			END_IF

		20:
			IF Executing THEN
				executeTime := executeTime + RTInfo_0.cycle_time / 1000;
			END_IF
			totalTime := totalTime + RTInfo_0.cycle_time / 1000;

			IF totalTime > 0 THEN
				Availability := UDINT_TO_REAL(executeTime) / UDINT_TO_REAL(totalTime) * 100;
			END_IF

			IF executeTime > 0 THEN
				Performance := LIMIT(0, IdealCycleTime * UDINT_TO_REAL(BadPortion + GoodPortion) / UDINT_TO_REAL(executeTime) * 100, 100);
			END_IF

			IF GoodPortion + BadPortion > 0 THEN
				Quality := UDINT_TO_REAL(GoodPortion) / UDINT_TO_REAL(GoodPortion + BadPortion) * 100;
			END_IF

			OEE := (Availability/100.0) * (Performance/100.0) * (Quality/100.0) * 100;

			IF Reset THEN
				executeTime := 0;
				totalTime := 0;
				GoodPortion := 0;
				BadPortion := 0;
			END_IF
	END_CASE

END_FUNCTION_BLOCK
```

### bottomFlapGlobal.typ
```iecst
TYPE
	gBottomFlapInterface_status_typ : 	STRUCT
		ready2 : BOOL;
		ready1 : BOOL;
		openCloseTime : UDINT;
		active : BOOL;
		waitingForNeighbour : BOOL;
		emptyReady : BOOL;
		approvedPortion : BOOL;
		neighbourWaiting : BOOL;
		neighbourDisappeared : BOOL;
		testResultFAT : BOOL; (*TRUE=good, FALSE=bad*)
	END_STRUCT;
	gBottomFlapInterface_para_typ : 	STRUCT
		brickStatus : gFlap_brick_status_typ;
		openTime : UDINT; (*Time the flap stays open*)
		flapTime : UDINT; (*Time that the flap is to open or close*)
		fallTime : UDINT; (*Time that a brick is to fall and be steady*)
		cassetteStartDelay : UDINT; (*Delay time of start cassette*)
		transmissionDelay : UDINT; (*Delay time of transmission to neighbour machine*)
		shaftMode : gBottomShaftMode_typ; (*Shaft mode can either be normal of empty*)
	END_STRUCT;
	gBottomFlapInterface_cmd_typ : 	STRUCT
		start1 : BOOL;
		start2 : BOOL;
		empty : BOOL;
		updateStatistics : BOOL;
		runFlapContinuously : BOOL;
		open : BOOL; (*Manuel mode to open flap from wing task.*)
		waitModeChange : BOOL; (*When changing to empty mode bottomFlap must wait a delay to make sure the 2 machines both have same mode.*)
		resetCassetteWaitTime : BOOL; (*Capcon -> bottomFlap. We teach a new brick please reset the wait time for cassette.*)
		brickStatusReady : BOOL;
		manuelMode : BOOL;
		wingTestManual : BOOL;
	END_STRUCT;
	gBottomFlapInterface_typ : 	STRUCT
		cmd : gBottomFlapInterface_cmd_typ;
		parameter : gBottomFlapInterface_para_typ;
		status : gBottomFlapInterface_status_typ;
	END_STRUCT;
	gBottomShaftMode_typ :
		(
		SHAFT_MODE_NORMAL, (*If shaft mode is normal then stage change to I070 where portion of items is transferred to bottom flap before waiting for cassette is ready *)
		SHAFT_MODE_EMPTY (*If shaft mode is empty then stage change to I100 where bottom flap is waiting for cassette is ready before portion of items is transferred to bottom flap *)
		);
END_TYPE
```

### bottomFlapGlobal.var
```iecst
VAR
	gBottomFlapInterface : gBottomFlapInterface_typ;
END_VAR
```

### Program Logical/modules/main/wing/cassette/cassette (IEC)

#### producing.st
```iecst
ACTION producing:

	CASE em.state OF

		STATE_STOPPED:
			interface.status.ready 		:= FALSE;
			em.cmd.sc 					:= TRUE;
			em.cmd.reset 				:= TRUE;

		STATE_IDLE:
			em.cmd.start := em.cmd.sc := TRUE;

		STATE_EXECUTE:

			CASE em.substate OF

				0:
					em.description := 'waiting for cassette to arrive';

					this.time.elapsed := 0;
					this.time.maximum := interface.parameter.cassetteDetectTime;
					IF NOT(this.hw.di_cassetteReady) THEN //casetteReady=FALSE means cassette is ready - Signal active low
						em.substate := 10;
					END_IF

				10:
					em.description := ' waiting for ready signal high in detect time';

					IF NOT(this.hw.di_cassetteReady) THEN //Cassette ready signal must still be FALSE
						this.time.elapsed	:= this.time.elapsed + em.status.cycleTime; //Casette signal must be stable for detect time (Works like a filter?)
						IF this.time.elapsed >= this.time.maximum THEN
							interface.status.ready 	:= TRUE;
							em.substate := 30;
						END_IF
					ELSE //Casette is no longer present
						em.substate := 0;
					END_IF

				30:
					em.description := 'waiting for start command';

					interface.status.ready := TRUE;

					IF interface.cmd.start <> interface.status.startAck THEN
						interface.status.ready 	:= FALSE;
						interface.status.dosing := FALSE;
						em.substate := 40;
					ELSIF interface.cmd.dosing AND NOT gBottomFlapInterface.status.approvedPortion AND NOT gBottomFlapInterface.status.neighbourDisappeared THEN
						interface.status.ready := FALSE;
						interface.status.dosing := TRUE;
						interface.status.startAck := interface.cmd.start - 1;
						interface.status.syncAck := interface.cmd.start - 1;
						em.substate := 40;
					ELSIF gMainInterface.line.bypassCassette AND this.hw.di_neighbourIsDosing THEN
						em.substate := 200;
					END_IF

				40:
					em.description := 'Wait for cassetteQueue to be free';

					IF this.hw.di_cassetteQueue THEN
						em.substate := 50;
					END_IF

				50:
					em.description := 'request to release cassette with other CM';

					IF gBottomFlapInterface.status.neighbourWaiting AND NOT this.hw.di_neighbourIsDosing AND NOT gBottomFlapInterface.status.approvedPortion THEN
						this.CassetteSync_0.Cancel := TRUE;
						this.CassetteSync_0.Request := FALSE;
					ELSE
						this.CassetteSync_0.Cancel := FALSE;
						this.CassetteSync_0.Request := TRUE;
					END_IF

					IF this.CassetteSync_0.Approved THEN
						this.CassetteSync_0.Request := FALSE;
						interface.status.syncAck := interface.cmd.start;
						em.substate := 70;
					ELSIF this.CassetteSync_0.CancelApproved THEN
						this.CassetteSync_0.Request := FALSE;
						this.CassetteSync_0.Cancel := FALSE;
						interface.status.syncAck := interface.cmd.start;
						interface.status.startAck := interface.cmd.start;
						em.substate := 30;
					END_IF

				70:
					em.description := 'waiting for cassette to leave sensor';

					this.hw.do_cassetteRelease := TRUE;

					IF this.hw.di_cassetteReady THEN
						this.time.elapsed := 0;
						this.time.maximum := interface.parameter.releaseTime;
						em.substate := 80;
					END_IF

				80:
					em.description := 'waiting for release time';

					this.time.elapsed := this.time.elapsed + em.status.cycleTime;
					IF this.time.elapsed >= this.time.maximum THEN
						this.hw.do_cassetteRelease 			:= FALSE;

						this.cassetteCounter := this.cassetteCounter + 1;
						interface.status.startAck := interface.cmd.start;
						em.substate := 0;
					END_IF

				200:
					em.description := 'Wait for cassetteQueue to be free';

					IF this.hw.di_cassetteQueue THEN
						em.substate := 210;
					END_IF

				210:
					em.description := 'waiting for cassette to leave sensor';

					this.hw.do_cassetteRelease := TRUE;

					IF this.hw.di_cassetteReady THEN
						this.time.elapsed := 0;
						this.time.maximum := interface.parameter.releaseTime;
						em.substate := 220;
					END_IF

				220:
					em.description := 'waiting for release time';

					this.time.elapsed := this.time.elapsed + em.status.cycleTime;
					IF this.time.elapsed >= this.time.maximum THEN
						this.hw.do_cassetteRelease 			:= FALSE;

						em.substate := 230;
					END_IF

				230:
					em.description := 'waiting for cassette to arrive';

					this.time.elapsed := 0;
					this.time.maximum := interface.parameter.cassetteDetectTime;
					IF NOT(this.hw.di_cassetteReady) THEN //casetteReady=FALSE means cassette is ready - Signal active low
						em.substate := 240;
					END_IF

				240:
					em.description := 'waiting for ready signal high in detect time';

					IF NOT(this.hw.di_cassetteReady) THEN //Cassette ready signal must still be FALSE
						this.time.elapsed	:= this.time.elapsed + em.status.cycleTime; //Casette signal must be stable for detect time (Works like a filter?)
						IF this.time.elapsed >= this.time.maximum THEN

							IF gMainInterface.line.bypassCassette AND this.hw.di_neighbourIsDosing THEN
								em.substate := 200;
							ELSE
								em.substate := 30;
							END_IF
						END_IF
					ELSE //Casette is no longer present
						em.substate := 230;
					END_IF

			END_CASE

			IF em.substate = 0 OR em.substate = 10 THEN
				this.statistics.waitForCassette := this.statistics.waitForCassette + (em.status.cycleTime / 1000);
			END_IF

			IF em.substate = 40 THEN
				this.statistics.cassetteQueue := this.statistics.cassetteQueue + (em.status.cycleTime / 1000);
			END_IF

			IF em.substate = 20 OR em.substate = 30 THEN
				this.statistics.waitForPortion := this.statistics.waitForPortion + (em.status.cycleTime / 1000);
			END_IF

			IF em.substate = 50 THEN
				this.statistics.waitForNeighbour := this.statistics.waitForNeighbour + (em.status.cycleTime / 1000);
			END_IF

			IF em.substate = 70 OR em.substate = 80 THEN
				this.statistics.realeaseCassette := this.statistics.realeaseCassette + (em.status.cycleTime / 1000);
			END_IF

		STATE_STOPPING,STATE_ABORTING,STATE_SUSPENDING:
			em.description 						:= 'stop all movement';
			this.hmi.status 					:= 1;
			interface.status.ready 				:= FALSE;
			this.hw.do_cassetteRelease 			:= FALSE;
			em.cmd.sc							:= TRUE;
			this.CassetteSync_0.Request 		:= FALSE;

		STATE_ABORTED, STATE_SUSPENDED:
			this.hmi.status 					:= 2;

			em.cmd.clear := em.state = STATE_ABORTED;
			em.cmd.start := em.state = STATE_SUSPENDED;
			em.cmd.sc := TRUE;

		STATE_CLEARING, STATE_UNSUSPENDING:
			brsmemset(ADR(this.alarm), 0, SIZEOF(this.alarm));

			em.cmd.sc := TRUE;

		ELSE
			em.cmd.sc := TRUE;

	END_CASE

END_ACTION
```

#### alarm.st
```iecst
ACTION alarm:

	// ALARM TO BE ADDED HERE...

END_ACTION
```

#### cassette.st - Init, cyclic, exit code
```iecst
PROGRAM _INIT

	em.setup.name 			:= 'cassette';
	em.setup.lastActivated	:= TRUE;

	setupPointers;

	interface.parameter.cassetteDetectTime := 10000;	// 10ms

	this.hwWu[0].do_active := TRUE;
	this.hwWu[1].do_active := TRUE;

END_PROGRAM

PROGRAM _CYCLIC

	setupPointers;
	ioMappingInput;

	CASE em.mode OF
		MODE_PRODUCING: producing;
		ELSE em.cmd.sc := TRUE;
	END_CASE

	em();

	this.CassetteSync_0.NeighbourActive 				:= this.hw.di_neighbourActive;
	this.CassetteSync_0.di_neighbourBricksInCassette 	:= this.hw.di_neighbourBricksInCassette;
	this.CassetteSync_0();
	IF this.hmi.do_bricksReadyInCassetteForce THEN
		this.hw.do_bricksReadyInCassette := TRUE;
	ELSE
		this.hw.do_bricksReadyInCassette 					:= this.CassetteSync_0.do_bricksReadyInCassette;
	END_IF

	IF this.hmi.do_dosingForce THEN
		this.hw.do_dosing := TRUE;
	ELSE
		this.hw.do_dosing := interface.cmd.dosing;
	END_IF
	this.CassetteUtilization_0.Enable 				:= gMainInterface.status.state = STATE_EXECUTE;
	this.CassetteUtilization_0.Substate 			:= em.substate;
	this.CassetteUtilization_0.CycleTime			:= em.status.cycleTime;
	this.CassetteUtilization_0.CassetteCounter 		:= this.cassetteCounter;
	this.CassetteUtilization_0.WaitingForNeighbour 	:= gBottomFlapInterface.status.waitingForNeighbour;
	this.CassetteUtilization_0();
	this.hmi.waitForPortion 				:= this.CassetteUtilization_0.WaitForPortion;
	this.hmi.releaseCassette 				:= this.CassetteUtilization_0.ReleaseCassette;
	this.hmi.waitForNeighbour 				:= this.CassetteUtilization_0.WaitForNeighbour;
	this.hmi.waitForQueue 					:= this.CassetteUtilization_0.WaitForQueue;
	this.hmi.waitForCassette 				:= this.CassetteUtilization_0.WaitForCassette;

	this.hmi.cycleTimeStopStation			:= this.CassetteUtilization_0.WaitForPortion+this.CassetteUtilization_0.ReleaseCassette+this.CassetteUtilization_0.WaitForNeighbour;
	this.hmi.cycleTime						:= this.CassetteUtilization_0.WaitForPortion+this.CassetteUtilization_0.ReleaseCassette;
	this.hmi.cassettesReleased 				:= this.CassetteUtilization_0.CassettesReleased;
	this.hmi.cassetteQueueSensor			:= NOT this.hw.di_cassetteQueue;
	this.hmi.cassetteReadySensor			:= NOT this.hw.di_cassetteReady;

	this.FlowMeasure_0.Enable := TRUE;
	this.FlowMeasure_0.CassetteQueue := this.hw.di_cassetteQueue;
	this.FlowMeasure_0.CassetteReady := this.hw.di_cassetteReady;
	this.FlowMeasure_0();

	// TOFF cassette signals (for PP99 linecontroller to avoid that signals gets lost in communication)
	this.TOF_cassetteReady.IN := this.hw.di_cassetteReady;
	this.TOF_cassetteReady.PT := gWingInterface.status.timeTOF_cassetteSignals;
	this.TOF_cassetteReady();
	this.TOF_cassetteQueue.IN := this.hw.di_cassetteQueue;
	this.TOF_cassetteQueue.PT := gWingInterface.status.timeTOF_cassetteSignals;
	this.TOF_cassetteQueue();

	this.hmi.di_cassetteReady_TOF := this.TOF_cassetteReady.Q;
	this.hmi.di_cassetteQueue_TOF := this.TOF_cassetteQueue.Q;

	// global interfacing
	gEthernetIPInterface.status.di_cassetteReady := this.hw.di_cassetteReady;
	gEthernetIPInterface.status.di_cassetteQueue := this.hw.di_cassetteQueue;
	gEthernetIPInterface.status.do_cassetteRelease := this.hw.do_cassetteRelease;

	// FAT test
	CASE testStateFAT OF

		0:
			IF interface.cmd.wingTestManual THEN

				IF this.hw.do_cassetteRelease=FALSE THEN
					this.oldCassetteReady := this.hw.di_cassetteReady;
					this.hw.do_cassetteRelease := TRUE;
					testStateFAT := 10;
				END_IF
			END_IF

		10:
			this.TON_test.IN := TRUE;
			this.TON_test.PT := T#1s;
			this.TON_test();

			IF this.TON_test.Q THEN
				this.TON_test.IN := FALSE;
				this.TON_test();
				// Test Fail
				interface.status.testResultFAT := FALSE;
				testStateFAT := 20;
			ELSIF this.oldCassetteReady <> this.hw.di_cassetteReady THEN
				this.TON_test.IN := FALSE;
				this.TON_test();
				// Test OK
				interface.status.testResultFAT := TRUE;
				testStateFAT := 20;
			END_IF

		20:
			// Test done go back
			this.hw.do_cassetteRelease := FALSE;
			interface.cmd.wingTestManual := FALSE;
			testStateFAT := 0;

	END_CASE

END_PROGRAM

PROGRAM _EXIT

END_PROGRAM
```

#### ioMappingInput.st
```iecst
ACTION ioMappingInput:

	IF this.hwWu[0].di_wingUnitActive THEN
		IF interface.cmd.cassetteIsBeingSimulated THEN
			this.hw.di_cassetteQueue			 := this.hwAir.di_cassetteQueue;
			this.hw.di_cassetteReady			 := this.hwAir.di_cassetteReady;
		ELSE
			this.hw.di_cassetteQueue			 := this.hwWu[0].di_cassetteQueue;
			this.hw.di_cassetteReady			 := this.hwWu[0].di_cassetteReady;
		END_IF
		this.hw.di_neighbourActive 			 := this.hwWu[0].di_neighbourActive;
		this.hw.di_neighbourIsDosing 		 := this.hwWu[0].di_neighbourIsDosing;
		this.hw.di_neighbourBricksInCassette := this.hwWu[0].di_neighbourBricksInCassette;
	ELSIF this.hwWu[1].di_wingUnitActive THEN
		IF interface.cmd.cassetteIsBeingSimulated THEN
			this.hw.di_cassetteQueue			 := this.hwAir.di_cassetteQueue;
			this.hw.di_cassetteReady			 := this.hwAir.di_cassetteReady;
		ELSE
			this.hw.di_cassetteQueue			 := this.hwWu[1].di_cassetteQueue;
			this.hw.di_cassetteReady			 := this.hwWu[1].di_cassetteReady;
		END_IF
		this.hw.di_neighbourActive 			 := this.hwWu[1].di_neighbourActive;
		this.hw.di_neighbourIsDosing 		 := this.hwWu[1].di_neighbourIsDosing;
		this.hw.di_neighbourBricksInCassette := this.hwWu[1].di_neighbourBricksInCassette;
	ELSE
		this.hw.di_cassetteQueue			 := this.hwAir.di_cassetteQueue;
		this.hw.di_cassetteReady			 := this.hwAir.di_cassetteReady;
		this.hw.di_neighbourActive 			 := this.hwAir.di_neighbourActive;
		this.hw.di_neighbourIsDosing 		 := this.hwAir.di_neighbourIsDosing;
		this.hw.di_neighbourBricksInCassette := this.hwAir.di_neighbourBricksInCassette;
	END_IF

END_ACTION
```

#### setupPointers.st
```iecst
ACTION setupPointers:
	interface ACCESS ADR(gCassetteInterface);
END_ACTION
```

#### local.typ - Local data types
```iecst
TYPE
	local_alarm_typ : 	STRUCT
		dummy : gAlarm_struct_typ;
	END_STRUCT;
	hmi_typ : 	STRUCT
		bottomNeighbourAccept : BOOL;
		status : USINT;
		waitForPortion : REAL;
		releaseCassette : REAL;
		waitForNeighbour : REAL;
		waitForQueue : REAL;
		waitForCassette : REAL;
		cycleTime : REAL;
		cycleTimeStopStation : REAL;
		cassettesReleased : UDINT;
		cassetteReadySensor : BOOL;
		cassetteQueueSensor : BOOL;
		di_cassetteReady_TOF : BOOL;
		di_cassetteQueue_TOF : BOOL;
		do_dosingForce : BOOL;
		do_bricksReadyInCassetteForce : BOOL;
	END_STRUCT;
	local_stat_typ : 	STRUCT
		realeaseCassette : UDINT;
		waitForCassette : UDINT;
		cassetteQueue : UDINT;
		waitForPortion : UDINT;
		waitForNeighbour : UDINT;
	END_STRUCT;
	local_typ : 	STRUCT
		hw : local_hw_typ;
		hwAir : local_hw_typ;
		hwWu : ARRAY[0..1]OF wu20_typ;
		hmi : hmi_typ;
		time : local_time_typ;
		alarm : local_alarm_typ;
		testSimCassetteReady : BOOL;
		TON_0 : TON;
		statistics : local_stat_typ;
		CassetteSync_0 : CassetteSync;
		CassetteUtilization_0 : CassetteUtilization;
		cassetteCounter : USINT;
		TOF_cassetteReady : TOF;
		TOF_cassetteQueue : TOF;
		FlowMeasure_0 : FlowMeasure;
		oldCassetteReady : BOOL;
		TON_test : TON;
	END_STRUCT;
	wu20_typ : 	STRUCT
		di_cassetteQueue : BOOL;
		di_neighbourActive : BOOL;
		di_cassetteReady : BOOL;
		di_neighbourIsDosing : BOOL;
		di_neighbourBricksInCassette : BOOL;
		do_active : BOOL; (*Alway true*)
		di_wingUnitActive : BOOL;
	END_STRUCT;
	local_hw_typ : 	STRUCT
		di_cassetteReady : BOOL; (*Signal name: DI_WU_CRDY
PJ95: WU_S
Connector: DI.15
Description: Signal from Shaft. Indicating a cassette is ready at the shaft. “0” indicates a cassette is ready*)
		di_cassetteQueue : BOOL; (*Signal name: DI_WU_CQUE
PJ95: WU_S
Connector: DI.14
Description: Signal from Shaft. Indicating a cassette queue on the transfer system after the CM. “0” indicates cassette queuing up.*)
		di_neighbourBricksInCassette : BOOL; (*Signal name: DI_WU_NCRDY
PJ95: WU_S
Connector: DI.17
Description: Signal from neighbour CM. “0” indicates elements from neighbour shaft are ready in cassette. Utilized for synchronization cassette stop with neighbour CM. Only relevant if DI_WU_NCON is active.*)
		do_cassetteRelease : BOOL; (*Signal name: DO_WU_CREL
PJ95: WU_S
Connector: DO.19
Description: Signal to shaft cassette stop. “1” means cassette is released*)
		do_bricksReadyInCassette : BOOL; (*Signal name: DO_WU_NCRDY
PJ95: WU_S
Connector: DO.17
Description: Signal to neighbour CM. “1” means elements from shaft are ready in cassette. Utilized for synchronization cassette stop with neighbour CM.*)
		di_neighbourActive : BOOL; (*Signal name: DI_WU_NCON
PJ95: WU_S
Connector: DI.18
Description: Signal from neighbour CM. “1” indicates a neighbour CM is connected and active.*)
		di_neighbourIsDosing : BOOL; (*Signal name: DI_WU_NDO
PJ95: WU_S
Connector: DI.08
Description: Signal from neighbour CM. “1” indicates a neighbour CM is dosing meaning empty cassettes are released. Only relevant if DI_WU_NCON is active*)
		do_dosing : BOOL; (*Signal name: DO_WU_NDO
PJ95: WU_S
Connector: DO.22
Description: Signal to neighbour CM. “1” indicates CM is dosing meaning empty cassettes are released*)
		do_testCassetteReady : BOOL;
	END_STRUCT;
END_TYPE
```

#### local.var - Local variables
```iecst
VAR
	this : {REDUND_UNREPLICABLE} local_typ;
	em : {REDUND_UNREPLICABLE} brdkEM;
	interface : REFERENCE TO gCassetteInterface_typ;
	testStateFAT : USINT;
END_VAR
```

#### LocalFunctions.fun
```iecst
{REDUND_ERROR} FUNCTION_BLOCK CassetteSync (*Function block that handles synchronization between two CMs*) (*$GROUP=User,$CAT=User,$GROUPICON=User.png,$CATICON=User.png*)
	VAR_INPUT
		Request : BOOL; (*Request synchronization with neighbour machine*)
		di_neighbourBricksInCassette : BOOL;
		NeighbourActive : BOOL;
		Cancel : BOOL;
	END_VAR
	VAR_OUTPUT
		do_bricksReadyInCassette : BOOL;
		Approved : BOOL; (*Syncronization with neighbour completed*)
		CancelApproved : BOOL;
	END_VAR
	VAR
		state : UINT;
		TON_timeout : TON;
		TON_transmissionDelay : TON;
	END_VAR
END_FUNCTION_BLOCK

FUNCTION_BLOCK CassetteUtilization
	VAR_INPUT
		Enable : BOOL;
		Substate : UINT;
		CycleTime : UDINT;
		WaitingForNeighbour : BOOL;
		CassetteCounter : UDINT;
	END_VAR
	VAR_OUTPUT
		CassettesReleased : UDINT;
		WaitForCassette : REAL;
		WaitForQueue : REAL;
		WaitForPortion : REAL;
		WaitForNeighbour : REAL;
		ReleaseCassette : REAL;
	END_VAR
	VAR
		state : UINT;
		_waitForCassette : UDINT;
		_waitForNeighbour : UDINT;
		_waitForPortion : UDINT;
		_waitForQueue : UDINT;
		_releaseCassette : UDINT;
		oldCassetteCounter : UDINT;
	END_VAR
END_FUNCTION_BLOCK

FUNCTION_BLOCK FallingEdgeTrigger
	VAR_INPUT
		start : BOOL;
		input : BOOL := FALSE;
	END_VAR
	VAR_OUTPUT
		output : BOOL;
	END_VAR
	VAR
		oldInput : BOOL;
		TON_timeout : TON;
	END_VAR
END_FUNCTION_BLOCK

FUNCTION_BLOCK FlowMeasure
	VAR_INPUT
		Enable : BOOL;
		CassetteReady : BOOL;
		CassetteQueue : BOOL;
	END_VAR
	VAR_OUTPUT
		FlowWaitTime : DINT;
		FlowQueueTime : DINT;
	END_VAR
	VAR
		state : INT;
		cassetteReadyTime : DINT;
		cassetteQueueTime : DINT;
	END_VAR
END_FUNCTION_BLOCK
```

#### LocalFunctions.st
```iecst
(* Function block that handles synchronization between two CMs *)
FUNCTION_BLOCK CassetteSync

	CASE state OF
		0:
			IF Request THEN
				do_bricksReadyInCassette := TRUE;
				state := 10;
			ELSIF Cancel THEN
				state := 220;
			END_IF

		10:
			IF di_neighbourBricksInCassette THEN
				state := 15;
			ELSIF Cancel THEN
				TON_timeout.IN := FALSE;
				TON_timeout();
				state := 200;
			END_IF

		15:
			TON_transmissionDelay.IN := TRUE;
			TON_transmissionDelay.PT:= T#10ms;
			TON_transmissionDelay();

			IF TON_transmissionDelay.Q THEN
				TON_transmissionDelay.IN := FALSE;
				TON_transmissionDelay();
				do_bricksReadyInCassette := FALSE;
				state := 20;
			END_IF

		20:
			IF NOT di_neighbourBricksInCassette THEN
				Approved := TRUE;
				state := 30;
			END_IF

		30:
			IF NOT Request THEN
				Approved := FALSE;
				state := 0;
			END_IF

		100:
			Approved := Request;

			IF NeighbourActive THEN
				Approved := FALSE;
				state := 0;
			END_IF

		200:
			do_bricksReadyInCassette := FALSE;

			TON_timeout.IN := TRUE;
			TON_timeout.PT := T#100ms;
			TON_timeout();

			IF di_neighbourBricksInCassette THEN
				TON_timeout.IN := FALSE;
				TON_timeout();
				state := 210;
			ELSIF TON_timeout.Q THEN
				TON_timeout.IN := FALSE;
				TON_timeout();
				state := 220;
			END_IF

		210:
			TON_timeout.IN := TRUE;
			TON_timeout.PT := T#100ms;
			TON_timeout();

			IF NOT di_neighbourBricksInCassette THEN
				TON_timeout.IN := FALSE;
				TON_timeout();
				Approved := TRUE;
				state := 30;
			ELSIF TON_timeout.Q THEN
				TON_timeout.IN := FALSE;
				TON_timeout();
				state := 220;
			END_IF

		220:
			CancelApproved := TRUE;

			IF NOT Cancel THEN
				CancelApproved := FALSE;
				state := 0;
			END_IF

	END_CASE

	IF NOT NeighbourActive THEN
		do_bricksReadyInCassette := FALSE;
		state := 100;
	END_IF

END_FUNCTION_BLOCK

FUNCTION_BLOCK FallingEdgeTrigger

	IF start THEN
		TON_timeout.IN := NOT output; // IF not output for 2s - timeout and make out=TRUE.
		TON_timeout.PT := T#2s;
		TON_timeout();

		IF (NOT input AND oldInput) OR TON_timeout.Q THEN
			TON_timeout(IN:=FALSE);
			output := TRUE;
		END_IF
		oldInput := input;

	ELSE
		TON_timeout(IN:=FALSE);
		output := oldInput := FALSE;
	END_IF

END_FUNCTION_BLOCK

FUNCTION_BLOCK CassetteUtilization

	CASE state OF
		0:
			IF Enable THEN
				state := 10;
			END_IF

		10:
			CASE Substate OF
				0,10:
					_waitForCassette := _waitForCassette + CycleTime;

				20,30:
					IF WaitingForNeighbour THEN
						_waitForNeighbour := _waitForNeighbour + CycleTime;
					ELSE
						_waitForPortion := _waitForPortion + CycleTime;
					END_IF

				40:
					_waitForQueue := _waitForQueue + CycleTime;

				50:
					_waitForNeighbour := _waitForNeighbour + CycleTime;

				70,80:
					_releaseCassette := _releaseCassette + CycleTime;
			END_CASE

	END_CASE

	IF CassetteCounter <> oldCassetteCounter THEN
		oldCassetteCounter := CassetteCounter;

		WaitForCassette := UDINT_TO_REAL(_waitForCassette)/1000;
		WaitForNeighbour :=  UDINT_TO_REAL(_waitForNeighbour)/1000;
		WaitForPortion :=  UDINT_TO_REAL(_waitForPortion)/1000;
		WaitForQueue :=  UDINT_TO_REAL(_waitForQueue)/1000;
		ReleaseCassette :=  UDINT_TO_REAL(_releaseCassette)/1000;

		CassettesReleased := CassetteCounter;

		_waitForCassette := 0;
		_waitForNeighbour := 0;
		_waitForPortion := 0;
		_waitForQueue := 0;
		_releaseCassette := 0;
	END_IF

	IF state <> 0 AND NOT Enable THEN
		state := 0;
	END_IF

END_FUNCTION_BLOCK

FUNCTION_BLOCK FlowMeasure

	CASE state OF
		0:
			IF Enable THEN
				state := 10;
			END_IF

		10:
			// Cassette wait
			IF CassetteReady AND cassetteReadyTime = 0 THEN
				cassetteReadyTime := TIME_TO_DINT(clock_ms());
			END_IF

			IF NOT CassetteReady AND cassetteReadyTime <> 0 THEN
				FlowWaitTime := TIME_TO_DINT(clock_ms()) - cassetteReadyTime;
				cassetteReadyTime := 0;
			END_IF

			IF cassetteReadyTime <> 0 AND FlowWaitTime + 2000 < TIME_TO_DINT(clock_ms()) - cassetteReadyTime THEN
				FlowWaitTime := TIME_TO_DINT(clock_ms()) - cassetteReadyTime;
			END_IF

			// Cassette queue
			IF NOT CassetteQueue AND cassetteQueueTime = 0 THEN
				cassetteQueueTime := TIME_TO_DINT(clock_ms());
			END_IF

			IF CassetteQueue AND cassetteQueueTime <> 0 THEN
				FlowQueueTime := TIME_TO_DINT(clock_ms()) - cassetteQueueTime;
				cassetteQueueTime := 0;
			END_IF

			IF cassetteQueueTime <> 0 AND FlowQueueTime + 2000 < TIME_TO_DINT(clock_ms()) - cassetteQueueTime THEN
				FlowQueueTime := TIME_TO_DINT(clock_ms()) - cassetteQueueTime;
			END_IF
	END_CASE

END_FUNCTION_BLOCK
```

### cassetteGlobal.typ
```iecst
TYPE
	gCassetteInterface_typ : 	STRUCT
		cmd : gCassetteInterface_cmd_typ;
		parameter : gCassetteInterface_parameter_typ;
		status : gCassetteInterface_status_typ;
	END_STRUCT;
	gCassetteInterface_cmd_typ : 	STRUCT
		start : UDINT;
		cassetteIsBeingSimulated : BOOL;
		dosing : BOOL;
		wingTestManual : BOOL;
	END_STRUCT;
	gCassetteInterface_status_typ : 	STRUCT
		ready : BOOL;
		startAck : UDINT;
		dosing : BOOL;
		syncAck : UDINT;
		testResultFAT : BOOL; (*TRUE=good, FALSE=bad*)
	END_STRUCT;
	gCassetteInterface_parameter_typ : 	STRUCT
		cassetteDetectTime : UDINT; (*Time that the cassette ready signal need to be low*)
		releaseTime : UDINT; (*Cassette release time*)
	END_STRUCT;
END_TYPE
```

### cassetteGlobal.var
```iecst
VAR
	gCassetteInterface : gCassetteInterface_typ;
END_VAR
```

### Package Logical/services/machine - This module is used to handle the machine configuration.

### Program Logical/services/machine/machine (IEC, version 1.00.0)
